  PROC DrawPart12()
    MoveL Offs(pOrigin,220.25,208.79,0.00),v40,z0,tPen\WObj:=wPaper;
    MoveL Offs(pOrigin,220.46,209.85,0.00),v40,fine,tPen\WObj:=wPaper;
    MoveL Offs(pOrigin,220.46,209.85,6.00),v60,z5,tPen\WObj:=wPaper;
    MoveL Offs(pOrigin,220.04,211.98,6.00),vTravel,z5,tPen\WObj:=wPaper;
    MoveL Offs(pOrigin,220.04,211.98,0.00),v60,z0,tPen\WObj:=wPaper;
    MoveL Offs(pOrigin,218.55,213.11,0.00),v40,z0,tPen\WObj:=wPaper;
    MoveL Offs(pOrigin,217.27,213.53,0.00),v40,z0,tPen\WObj:=wPaper;
    MoveL Offs(pOrigin,216.64,214.74,0.00),v40,z0,tPen\WObj:=wPaper;
    MoveL Offs(pOrigin,212.39,219.62,0.00),v40,z0,tPen\WObj:=wPaper;
    MoveL Offs(pOrigin,210.40,223.02,0.00),v40,z0,tPen\WObj:=wPaper;
    MoveL Offs(pOrigin,208.35,227.70,0.00),v40,fine,tPen\WObj:=wPaper;
    MoveL Offs(pOrigin,208.35,227.70,6.00),v60,z5,tPen\WObj:=wPaper;
    MoveL Offs(pOrigin,209.84,224.09,6.00),vTravel,z5,tPen\WObj:=wPaper;
    MoveL Offs(pOrigin,209.84,224.09,0.00),v60,z0,tPen\WObj:=wPaper;
    MoveL Offs(pOrigin,209.62,224.51,0.00),v40,z0,tPen\WObj:=wPaper;
    MoveL Offs(pOrigin,209.84,224.09,0.00),v40,fine,tPen\WObj:=wPaper;
    MoveL Offs(pOrigin,209.84,224.09,6.00),v60,z5,tPen\WObj:=wPaper;
    MoveL Offs(pOrigin,211.32,221.11,6.00),vTravel,z5,tPen\WObj:=wPaper;
    MoveL Offs(pOrigin,211.32,221.11,0.00),v60,z0,tPen\WObj:=wPaper;
    MoveL Offs(pOrigin,211.11,221.54,0.00),v40,z0,tPen\WObj:=wPaper;
    MoveL Offs(pOrigin,211.32,221.11,0.00),v40,fine,tPen\WObj:=wPaper;
    MoveL Offs(pOrigin,211.32,221.11,6.00),v60,z5,tPen\WObj:=wPaper;
    MoveL Offs(pOrigin,217.06,213.46,6.00),vTravel,z5,tPen\WObj:=wPaper;
    MoveL Offs(pOrigin,217.06,213.46,0.00),v60,z0,tPen\WObj:=wPaper;
    MoveL Offs(pOrigin,216.43,212.82,0.00),v40,fine,tPen\WObj:=wPaper;
    MoveL Offs(pOrigin,216.43,212.82,6.00),v60,z5,tPen\WObj:=wPaper;
    MoveL Offs(pOrigin,220.04,211.98,6.00),vTravel,z5,tPen\WObj:=wPaper;
    MoveL Offs(pOrigin,220.04,211.98,0.00),v60,z0,tPen\WObj:=wPaper;
    MoveL Offs(pOrigin,221.74,211.62,0.00),v40,z0,tPen\WObj:=wPaper;
    MoveL Offs(pOrigin,226.62,209.21,0.00),v40,fine,tPen\WObj:=wPaper;
    MoveL Offs(pOrigin,226.62,209.21,6.00),v60,z5,tPen\WObj:=wPaper;
    MoveL Offs(pOrigin,223.44,207.51,6.00),vTravel,z5,tPen\WObj:=wPaper;
    MoveL Offs(pOrigin,223.44,207.51,0.00),v60,z0,tPen\WObj:=wPaper;
    MoveL Offs(pOrigin,221.95,209.00,0.00),v40,z0,tPen\WObj:=wPaper;
    MoveL Offs(pOrigin,223.44,207.51,0.00),v40,fine,tPen\WObj:=wPaper;
    MoveL Offs(pOrigin,223.44,207.51,6.00),v60,z5,tPen\WObj:=wPaper;
    MoveL Offs(pOrigin,225.35,205.60,6.00),vTravel,z5,tPen\WObj:=wPaper;
    MoveL Offs(pOrigin,225.35,205.60,0.00),v60,z0,tPen\WObj:=wPaper;
    MoveL Offs(pOrigin,223.65,207.30,0.00),v40,z0,tPen\WObj:=wPaper;
    MoveL Offs(pOrigin,225.35,205.60,0.00),v40,fine,tPen\WObj:=wPaper;
    MoveL Offs(pOrigin,225.35,205.60,6.00),v60,z5,tPen\WObj:=wPaper;
    MoveL Offs(pOrigin,227.05,203.69,6.00),vTravel,z5,tPen\WObj:=wPaper;
    MoveL Offs(pOrigin,227.05,203.69,0.00),v60,z0,tPen\WObj:=wPaper;
    MoveL Offs(pOrigin,221.67,209.57,0.00),v40,z0,tPen\WObj:=wPaper;
    MoveL Offs(pOrigin,220.53,210.06,0.00),v40,z0,tPen\WObj:=wPaper;
    MoveL Offs(pOrigin,220.04,210.91,0.00),v40,z0,tPen\WObj:=wPaper;
    MoveL Offs(pOrigin,220.04,211.98,0.00),v40,fine,tPen\WObj:=wPaper;
    MoveL Offs(pOrigin,220.04,211.98,6.00),v60,z5,tPen\WObj:=wPaper;
    MoveL Offs(pOrigin,213.52,208.93,6.00),vTravel,z5,tPen\WObj:=wPaper;
    MoveL Offs(pOrigin,213.52,208.93,0.00),v60,z0,tPen\WObj:=wPaper;
    MoveL Offs(pOrigin,215.57,210.91,0.00),v40,z0,tPen\WObj:=wPaper;
    MoveL Offs(pOrigin,213.52,208.93,0.00),v40,fine,tPen\WObj:=wPaper;
    MoveL Offs(pOrigin,213.52,208.93,6.00),v60,z5,tPen\WObj:=wPaper;
    MoveL Offs(pOrigin,210.69,206.88,6.00),vTravel,z5,tPen\WObj:=wPaper;
    MoveL Offs(pOrigin,210.69,206.88,0.00),v60,z0,tPen\WObj:=wPaper;
    MoveL Offs(pOrigin,210.26,205.18,0.00),v40,z0,tPen\WObj:=wPaper;
    MoveL Offs(pOrigin,197.94,190.73,0.00),v40,z0,tPen\WObj:=wPaper;
    MoveL Offs(pOrigin,197.51,189.88,0.00),v40,z0,tPen\WObj:=wPaper;
    MoveL Offs(pOrigin,197.73,189.24,0.00),v40,z0,tPen\WObj:=wPaper;
    MoveL Offs(pOrigin,207.93,185.41,0.00),v40,z0,tPen\WObj:=wPaper;
    MoveL Offs(pOrigin,208.77,185.41,0.00),v40,z0,tPen\WObj:=wPaper;
    MoveL Offs(pOrigin,213.24,188.18,0.00),v40,z0,tPen\WObj:=wPaper;
    MoveL Offs(pOrigin,220.68,194.98,0.00),v40,z0,tPen\WObj:=wPaper;
    MoveL Offs(pOrigin,222.38,195.82,0.00),v40,fine,tPen\WObj:=wPaper;
    MoveL Offs(pOrigin,222.38,195.82,6.00),v60,z5,tPen\WObj:=wPaper;
    MoveL Offs(pOrigin,217.13,191.50,6.00),vTravel,z5,tPen\WObj:=wPaper;
    MoveL Offs(pOrigin,217.13,191.50,0.00),v60,z0,tPen\WObj:=wPaper;
    MoveL Offs(pOrigin,218.98,193.27,0.00),v40,z0,tPen\WObj:=wPaper;
    MoveL Offs(pOrigin,217.13,191.50,0.00),v40,fine,tPen\WObj:=wPaper;
    MoveL Offs(pOrigin,217.13,191.50,6.00),v60,z5,tPen\WObj:=wPaper;
    MoveL Offs(pOrigin,215.36,189.88,6.00),vTravel,z5,tPen\WObj:=wPaper;
    MoveL Offs(pOrigin,215.36,189.88,0.00),v60,z0,tPen\WObj:=wPaper;
    MoveL Offs(pOrigin,216.21,190.73,0.00),v40,z0,tPen\WObj:=wPaper;
    MoveL Offs(pOrigin,215.36,189.88,0.00),v40,fine,tPen\WObj:=wPaper;
    MoveL Offs(pOrigin,215.36,189.88,6.00),v60,z5,tPen\WObj:=wPaper;
    MoveL Offs(pOrigin,207.93,185.20,6.00),vTravel,z5,tPen\WObj:=wPaper;
    MoveL Offs(pOrigin,207.93,185.20,0.00),v60,z0,tPen\WObj:=wPaper;
    MoveL Offs(pOrigin,207.50,184.56,0.00),v40,z0,tPen\WObj:=wPaper;
    MoveL Offs(pOrigin,195.60,178.26,0.00),v40,z0,tPen\WObj:=wPaper;
    MoveL Offs(pOrigin,194.68,177.55,0.00),v40,z0,tPen\WObj:=wPaper;
    MoveL Offs(pOrigin,194.54,176.49,0.00),v40,z0,tPen\WObj:=wPaper;
    MoveL Offs(pOrigin,201.76,148.65,0.00),v40,z0,tPen\WObj:=wPaper;
    MoveL Offs(pOrigin,207.07,129.74,0.00),v40,z0,tPen\WObj:=wPaper;
    MoveL Offs(pOrigin,208.14,124.85,0.00),v40,z0,tPen\WObj:=wPaper;
    MoveL Offs(pOrigin,207.71,123.36,0.00),v40,z0,tPen\WObj:=wPaper;
    MoveL Offs(pOrigin,207.71,121.66,0.00),v40,z0,tPen\WObj:=wPaper;
    MoveL Offs(pOrigin,208.77,114.01,0.00),v40,z0,tPen\WObj:=wPaper;
    MoveL Offs(pOrigin,210.48,95.53,0.00),v40,fine,tPen\WObj:=wPaper;
    MoveL Offs(pOrigin,210.48,95.53,6.00),v60,z5,tPen\WObj:=wPaper;
    MoveL Offs(pOrigin,230.02,83.20,6.00),vTravel,z5,tPen\WObj:=wPaper;
    MoveL Offs(pOrigin,230.02,83.20,0.00),v60,z0,tPen\WObj:=wPaper;
    MoveL Offs(pOrigin,230.95,82.56,0.00),v40,z0,tPen\WObj:=wPaper;
    MoveL Offs(pOrigin,233.57,77.46,0.00),v40,z0,tPen\WObj:=wPaper;
    MoveL Offs(pOrigin,236.82,73.00,0.00),v40,z0,tPen\WObj:=wPaper;
    MoveL Offs(pOrigin,236.40,73.43,0.00),v40,z0,tPen\WObj:=wPaper;
    MoveL Offs(pOrigin,236.19,73.85,0.00),v40,z0,tPen\WObj:=wPaper;
    MoveL Offs(pOrigin,236.40,73.43,0.00),v40,fine,tPen\WObj:=wPaper;
    MoveL Offs(pOrigin,236.40,73.43,6.00),v60,z5,tPen\WObj:=wPaper;
    MoveL Offs(pOrigin,235.34,63.22,6.00),vTravel,z5,tPen\WObj:=wPaper;
    MoveL Offs(pOrigin,235.34,63.22,0.00),v60,z0,tPen\WObj:=wPaper;
    MoveL Offs(pOrigin,230.88,66.06,0.00),v40,z0,tPen\WObj:=wPaper;
    MoveL Offs(pOrigin,227.69,67.26,0.00),v40,z0,tPen\WObj:=wPaper;
    MoveL Offs(pOrigin,226.84,67.26,0.00),v40,fine,tPen\WObj:=wPaper;
    MoveL Offs(pOrigin,226.84,67.26,6.00),v60,z5,tPen\WObj:=wPaper;
    MoveL Offs(pOrigin,226.62,65.99,6.00),vTravel,z5,tPen\WObj:=wPaper;
    MoveL Offs(pOrigin,226.62,65.99,0.00),v60,z0,tPen\WObj:=wPaper;
    MoveL Offs(pOrigin,228.04,64.71,0.00),v40,z0,tPen\WObj:=wPaper;
    MoveL Offs(pOrigin,235.12,54.09,0.00),v40,z0,tPen\WObj:=wPaper;
    MoveL Offs(pOrigin,234.70,54.51,0.00),v40,z0,tPen\WObj:=wPaper;
    MoveL Offs(pOrigin,234.49,54.94,0.00),v40,z0,tPen\WObj:=wPaper;
    MoveL Offs(pOrigin,234.70,54.51,0.00),v40,fine,tPen\WObj:=wPaper;
    MoveL Offs(pOrigin,234.70,54.51,6.00),v60,z5,tPen\WObj:=wPaper;
    MoveL Offs(pOrigin,238.74,39.85,6.00),vTravel,z5,tPen\WObj:=wPaper;
    MoveL Offs(pOrigin,238.74,39.85,0.00),v60,z0,tPen\WObj:=wPaper;
    MoveL Offs(pOrigin,242.14,39.64,0.00),v40,z0,tPen\WObj:=wPaper;
    MoveL Offs(pOrigin,242.14,39.64,0.00),v40,z0,tPen\WObj:=wPaper;
    MoveL Offs(pOrigin,241.93,37.30,0.00),v40,z0,tPen\WObj:=wPaper;
    MoveL Offs(pOrigin,242.70,35.60,0.00),v40,z0,tPen\WObj:=wPaper;
    MoveL Offs(pOrigin,243.62,34.82,0.00),v40,z0,tPen\WObj:=wPaper;
    MoveL Offs(pOrigin,244.69,34.75,0.00),v40,z0,tPen\WObj:=wPaper;
  ENDPROC

  PROC DrawPart13()
    MoveL Offs(pOrigin,244.69,34.75,0.00),v40,z0,tPen\WObj:=wPaper;
    MoveL Offs(pOrigin,245.25,36.24,0.00),v40,z0,tPen\WObj:=wPaper;
    MoveL Offs(pOrigin,246.81,38.15,0.00),v40,z0,tPen\WObj:=wPaper;
    MoveL Offs(pOrigin,254.25,44.10,0.00),v40,z0,tPen\WObj:=wPaper;
    MoveL Offs(pOrigin,264.45,51.18,0.00),v40,z0,tPen\WObj:=wPaper;
    MoveL Offs(pOrigin,270.19,53.80,0.00),v40,z0,tPen\WObj:=wPaper;
    MoveL Offs(pOrigin,270.61,54.30,0.00),v40,z0,tPen\WObj:=wPaper;
    MoveL Offs(pOrigin,270.61,54.30,0.00),v40,z0,tPen\WObj:=wPaper;
    MoveL Offs(pOrigin,269.62,57.28,0.00),v40,z0,tPen\WObj:=wPaper;
    MoveL Offs(pOrigin,268.20,59.40,0.00),v40,z0,tPen\WObj:=wPaper;
    MoveL Offs(pOrigin,266.36,61.10,0.00),v40,fine,tPen\WObj:=wPaper;
    MoveL Offs(pOrigin,266.36,61.10,6.00),v60,z5,tPen\WObj:=wPaper;
    MoveL Offs(pOrigin,267.42,61.74,6.00),vTravel,z5,tPen\WObj:=wPaper;
    MoveL Offs(pOrigin,267.42,61.74,0.00),v60,z0,tPen\WObj:=wPaper;
    MoveL Offs(pOrigin,269.12,59.83,0.00),v40,z0,tPen\WObj:=wPaper;
    MoveL Offs(pOrigin,270.68,57.28,0.00),v40,z0,tPen\WObj:=wPaper;
    MoveL Offs(pOrigin,271.25,54.94,0.00),v40,z0,tPen\WObj:=wPaper;
    MoveL Offs(pOrigin,270.61,54.30,0.00),v40,z0,tPen\WObj:=wPaper;
    MoveL Offs(pOrigin,271.25,54.51,0.00),v40,z0,tPen\WObj:=wPaper;
    MoveL Offs(pOrigin,272.10,54.51,0.00),v40,z0,tPen\WObj:=wPaper;
    MoveL Offs(pOrigin,273.16,55.15,0.00),v40,z0,tPen\WObj:=wPaper;
    MoveL Offs(pOrigin,273.16,55.15,0.00),v40,z0,tPen\WObj:=wPaper;
    MoveL Offs(pOrigin,271.11,59.83,0.00),v40,z0,tPen\WObj:=wPaper;
    MoveL Offs(pOrigin,269.55,61.31,0.00),v40,fine,tPen\WObj:=wPaper;
    MoveL Offs(pOrigin,269.55,61.31,6.00),v60,z5,tPen\WObj:=wPaper;
    MoveL Offs(pOrigin,271.04,61.31,6.00),vTravel,z5,tPen\WObj:=wPaper;
    MoveL Offs(pOrigin,271.04,61.31,0.00),v60,z0,tPen\WObj:=wPaper;
    MoveL Offs(pOrigin,270.83,61.74,0.00),v40,z0,tPen\WObj:=wPaper;
    MoveL Offs(pOrigin,271.04,61.31,0.00),v40,z0,tPen\WObj:=wPaper;
    MoveL Offs(pOrigin,271.67,60.67,0.00),v40,z0,tPen\WObj:=wPaper;
    MoveL Offs(pOrigin,271.46,61.10,0.00),v40,z0,tPen\WObj:=wPaper;
    MoveL Offs(pOrigin,271.67,60.67,0.00),v40,fine,tPen\WObj:=wPaper;
    MoveL Offs(pOrigin,271.67,60.67,6.00),v60,z5,tPen\WObj:=wPaper;
    MoveL Offs(pOrigin,272.31,59.61,6.00),vTravel,z5,tPen\WObj:=wPaper;
    MoveL Offs(pOrigin,272.31,59.61,0.00),v60,z0,tPen\WObj:=wPaper;
    MoveL Offs(pOrigin,272.10,60.04,0.00),v40,z0,tPen\WObj:=wPaper;
    MoveL Offs(pOrigin,272.31,59.61,0.00),v40,fine,tPen\WObj:=wPaper;
    MoveL Offs(pOrigin,272.31,59.61,6.00),v60,z5,tPen\WObj:=wPaper;
    MoveL Offs(pOrigin,270.61,57.06,6.00),vTravel,z5,tPen\WObj:=wPaper;
    MoveL Offs(pOrigin,270.61,57.06,0.00),v60,z0,tPen\WObj:=wPaper;
    MoveL Offs(pOrigin,270.40,57.49,0.00),v40,z0,tPen\WObj:=wPaper;
    MoveL Offs(pOrigin,270.61,57.06,0.00),v40,z0,tPen\WObj:=wPaper;
    MoveL Offs(pOrigin,269.55,57.06,0.00),v40,z0,tPen\WObj:=wPaper;
    MoveL Offs(pOrigin,269.34,57.49,0.00),v40,z0,tPen\WObj:=wPaper;
    MoveL Offs(pOrigin,269.55,57.06,0.00),v40,fine,tPen\WObj:=wPaper;
    MoveL Offs(pOrigin,269.55,57.06,6.00),v60,z5,tPen\WObj:=wPaper;
    MoveL Offs(pOrigin,267.85,59.83,6.00),vTravel,z5,tPen\WObj:=wPaper;
    MoveL Offs(pOrigin,267.85,59.83,0.00),v60,z0,tPen\WObj:=wPaper;
    MoveL Offs(pOrigin,268.06,59.40,0.00),v40,z0,tPen\WObj:=wPaper;
    MoveL Offs(pOrigin,267.85,59.83,0.00),v40,fine,tPen\WObj:=wPaper;
    MoveL Offs(pOrigin,267.85,59.83,6.00),v60,z5,tPen\WObj:=wPaper;
    MoveL Offs(pOrigin,270.19,62.80,6.00),vTravel,z5,tPen\WObj:=wPaper;
    MoveL Offs(pOrigin,270.19,62.80,0.00),v60,z0,tPen\WObj:=wPaper;
    MoveL Offs(pOrigin,268.27,62.45,0.00),v40,z0,tPen\WObj:=wPaper;
    MoveL Offs(pOrigin,266.15,61.17,0.00),v40,z0,tPen\WObj:=wPaper;
    MoveL Offs(pOrigin,264.24,60.53,0.00),v40,z0,tPen\WObj:=wPaper;
    MoveL Offs(pOrigin,261.26,59.05,0.00),v40,z0,tPen\WObj:=wPaper;
    MoveL Offs(pOrigin,257.86,56.64,0.00),v40,z0,tPen\WObj:=wPaper;
    MoveL Offs(pOrigin,248.94,47.92,0.00),v40,z0,tPen\WObj:=wPaper;
    MoveL Offs(pOrigin,245.32,43.67,0.00),v40,z0,tPen\WObj:=wPaper;
    MoveL Offs(pOrigin,242.77,40.06,0.00),v40,z0,tPen\WObj:=wPaper;
    MoveL Offs(pOrigin,242.14,39.64,0.00),v40,fine,tPen\WObj:=wPaper;
    MoveL Offs(pOrigin,242.14,39.64,6.00),v60,z5,tPen\WObj:=wPaper;
    MoveL Offs(pOrigin,246.18,37.30,6.00),vTravel,z5,tPen\WObj:=wPaper;
    MoveL Offs(pOrigin,246.18,37.30,0.00),v60,z0,tPen\WObj:=wPaper;
    MoveL Offs(pOrigin,247.02,38.15,0.00),v40,z0,tPen\WObj:=wPaper;
    MoveL Offs(pOrigin,246.18,37.30,0.00),v40,fine,tPen\WObj:=wPaper;
    MoveL Offs(pOrigin,246.18,37.30,6.00),v60,z5,tPen\WObj:=wPaper;
    MoveL Offs(pOrigin,247.88,38.79,6.00),vTravel,z5,tPen\WObj:=wPaper;
    MoveL Offs(pOrigin,247.88,38.79,0.00),v60,z0,tPen\WObj:=wPaper;
    MoveL Offs(pOrigin,248.30,39.21,0.00),v40,z0,tPen\WObj:=wPaper;
    MoveL Offs(pOrigin,247.88,38.79,0.00),v40,fine,tPen\WObj:=wPaper;
    MoveL Offs(pOrigin,247.88,38.79,6.00),v60,z5,tPen\WObj:=wPaper;
    MoveL Offs(pOrigin,249.15,39.85,6.00),vTravel,z5,tPen\WObj:=wPaper;
    MoveL Offs(pOrigin,249.15,39.85,0.00),v60,z0,tPen\WObj:=wPaper;
    MoveL Offs(pOrigin,250.00,40.70,0.00),v40,z0,tPen\WObj:=wPaper;
    MoveL Offs(pOrigin,249.15,39.85,0.00),v40,fine,tPen\WObj:=wPaper;
    MoveL Offs(pOrigin,249.15,39.85,6.00),v60,z5,tPen\WObj:=wPaper;
    MoveL Offs(pOrigin,244.69,34.75,6.00),vTravel,z5,tPen\WObj:=wPaper;
    MoveL Offs(pOrigin,244.69,34.75,0.00),v60,z0,tPen\WObj:=wPaper;
    MoveL Offs(pOrigin,244.69,33.47,0.00),v40,z0,tPen\WObj:=wPaper;
    MoveL Offs(pOrigin,245.75,31.42,0.00),v40,z0,tPen\WObj:=wPaper;
    MoveL Offs(pOrigin,247.45,30.50,0.00),v40,z0,tPen\WObj:=wPaper;
    MoveL Offs(pOrigin,249.79,30.50,0.00),v40,z0,tPen\WObj:=wPaper;
    MoveL Offs(pOrigin,250.43,30.08,0.00),v40,z0,tPen\WObj:=wPaper;
    MoveL Offs(pOrigin,250.43,30.08,0.00),v40,z0,tPen\WObj:=wPaper;
    MoveL Offs(pOrigin,249.57,29.15,0.00),v40,z0,tPen\WObj:=wPaper;
    MoveL Offs(pOrigin,215.15,21.79,0.00),v40,z0,tPen\WObj:=wPaper;
    MoveL Offs(pOrigin,211.54,20.51,0.00),v40,z0,tPen\WObj:=wPaper;
    MoveL Offs(pOrigin,210.05,20.73,0.00),v40,z0,tPen\WObj:=wPaper;
    MoveL Offs(pOrigin,210.05,20.73,0.00),v40,z0,tPen\WObj:=wPaper;
    MoveL Offs(pOrigin,210.05,21.15,0.00),v40,z0,tPen\WObj:=wPaper;
    MoveL Offs(pOrigin,209.41,21.36,0.00),v40,z0,tPen\WObj:=wPaper;
    MoveL Offs(pOrigin,208.56,20.94,0.00),v40,fine,tPen\WObj:=wPaper;
    MoveL Offs(pOrigin,208.56,20.94,6.00),v60,z5,tPen\WObj:=wPaper;
    MoveL Offs(pOrigin,210.05,20.73,6.00),vTravel,z5,tPen\WObj:=wPaper;
    MoveL Offs(pOrigin,210.05,20.73,0.00),v60,z0,tPen\WObj:=wPaper;
    MoveL Offs(pOrigin,208.99,18.39,0.00),v40,z0,tPen\WObj:=wPaper;
    MoveL Offs(pOrigin,209.06,17.33,0.00),v40,z0,tPen\WObj:=wPaper;
    MoveL Offs(pOrigin,209.41,17.11,0.00),v40,z0,tPen\WObj:=wPaper;
    MoveL Offs(pOrigin,233.43,14.99,0.00),v40,z0,tPen\WObj:=wPaper;
    MoveL Offs(pOrigin,274.86,25.83,0.00),v40,fine,tPen\WObj:=wPaper;
    MoveL Offs(pOrigin,274.86,25.83,6.00),v60,z5,tPen\WObj:=wPaper;
    MoveL Offs(pOrigin,273.80,27.74,6.00),vTravel,z5,tPen\WObj:=wPaper;
    MoveL Offs(pOrigin,273.80,27.74,0.00),v60,z0,tPen\WObj:=wPaper;
    MoveL Offs(pOrigin,234.27,17.96,0.00),v40,z0,tPen\WObj:=wPaper;
    MoveL Offs(pOrigin,231.30,17.96,0.00),v40,z0,tPen\WObj:=wPaper;
    MoveL Offs(pOrigin,212.60,19.88,0.00),v40,z0,tPen\WObj:=wPaper;
    MoveL Offs(pOrigin,211.96,20.51,0.00),v40,fine,tPen\WObj:=wPaper;
    MoveL Offs(pOrigin,211.96,20.51,6.00),v60,z5,tPen\WObj:=wPaper;
    MoveL Offs(pOrigin,208.99,17.11,6.00),vTravel,z5,tPen\WObj:=wPaper;
    MoveL Offs(pOrigin,208.99,17.11,0.00),v60,z0,tPen\WObj:=wPaper;
    MoveL Offs(pOrigin,208.77,16.26,0.00),v40,z0,tPen\WObj:=wPaper;
    MoveL Offs(pOrigin,209.41,14.35,0.00),v40,fine,tPen\WObj:=wPaper;
    MoveL Offs(pOrigin,209.41,14.35,6.00),v60,z5,tPen\WObj:=wPaper;
    MoveL Offs(pOrigin,207.07,13.93,6.00),vTravel,z5,tPen\WObj:=wPaper;
    MoveL Offs(pOrigin,207.07,13.93,0.00),v60,z0,tPen\WObj:=wPaper;
    MoveL Offs(pOrigin,208.99,13.78,0.00),v40,z0,tPen\WObj:=wPaper;
    MoveL Offs(pOrigin,209.84,14.35,0.00),v40,z0,tPen\WObj:=wPaper;
    MoveL Offs(pOrigin,212.81,14.35,0.00),v40,z0,tPen\WObj:=wPaper;
  ENDPROC

  PROC DrawPart14()
    MoveL Offs(pOrigin,232.15,12.23,0.00),v40,z0,tPen\WObj:=wPaper;
    MoveL Offs(pOrigin,235.12,12.44,0.00),v40,z0,tPen\WObj:=wPaper;
    MoveL Offs(pOrigin,276.35,23.27,0.00),v40,z0,tPen\WObj:=wPaper;
    MoveL Offs(pOrigin,276.56,23.70,0.00),v40,fine,tPen\WObj:=wPaper;
    MoveL Offs(pOrigin,276.56,23.70,6.00),v60,z5,tPen\WObj:=wPaper;
    MoveL Offs(pOrigin,273.59,29.01,6.00),vTravel,z5,tPen\WObj:=wPaper;
    MoveL Offs(pOrigin,273.59,29.01,0.00),v60,z0,tPen\WObj:=wPaper;
    MoveL Offs(pOrigin,272.31,29.01,0.00),v40,z0,tPen\WObj:=wPaper;
    MoveL Offs(pOrigin,271.89,29.44,0.00),v40,z0,tPen\WObj:=wPaper;
    MoveL Offs(pOrigin,271.89,29.44,0.00),v40,z0,tPen\WObj:=wPaper;
    MoveL Offs(pOrigin,272.31,30.08,0.00),v40,z0,tPen\WObj:=wPaper;
    MoveL Offs(pOrigin,273.59,30.08,0.00),v40,z0,tPen\WObj:=wPaper;
    MoveL Offs(pOrigin,273.59,30.08,0.00),v40,z0,tPen\WObj:=wPaper;
    MoveL Offs(pOrigin,274.01,30.50,0.00),v40,z0,tPen\WObj:=wPaper;
    MoveL Offs(pOrigin,282.94,33.62,0.00),v40,z0,tPen\WObj:=wPaper;
    MoveL Offs(pOrigin,285.91,35.39,0.00),v40,z0,tPen\WObj:=wPaper;
    MoveL Offs(pOrigin,285.91,35.39,0.00),v40,z0,tPen\WObj:=wPaper;
    MoveL Offs(pOrigin,287.83,35.74,0.00),v40,z0,tPen\WObj:=wPaper;
    MoveL Offs(pOrigin,288.25,36.45,0.00),v40,z0,tPen\WObj:=wPaper;
    MoveL Offs(pOrigin,288.46,36.45,0.00),v40,z0,tPen\WObj:=wPaper;
    MoveL Offs(pOrigin,290.80,37.37,0.00),v40,z0,tPen\WObj:=wPaper;
    MoveL Offs(pOrigin,291.51,38.36,0.00),v40,z0,tPen\WObj:=wPaper;
    MoveL Offs(pOrigin,291.65,39.42,0.00),v40,z0,tPen\WObj:=wPaper;
    MoveL Offs(pOrigin,289.60,45.59,0.00),v40,z0,tPen\WObj:=wPaper;
    MoveL Offs(pOrigin,288.67,46.22,0.00),v40,z0,tPen\WObj:=wPaper;
    MoveL Offs(pOrigin,287.61,46.22,0.00),v40,z0,tPen\WObj:=wPaper;
    MoveL Offs(pOrigin,284.42,45.02,0.00),v40,z0,tPen\WObj:=wPaper;
    MoveL Offs(pOrigin,283.79,44.10,0.00),v40,z0,tPen\WObj:=wPaper;
    MoveL Offs(pOrigin,285.70,39.21,0.00),v40,z0,tPen\WObj:=wPaper;
    MoveL Offs(pOrigin,285.98,36.88,0.00),v40,z0,tPen\WObj:=wPaper;
    MoveL Offs(pOrigin,288.46,36.45,0.00),v40,fine,tPen\WObj:=wPaper;
    MoveL Offs(pOrigin,288.46,36.45,6.00),v60,z5,tPen\WObj:=wPaper;
    MoveL Offs(pOrigin,287.40,38.58,6.00),vTravel,z5,tPen\WObj:=wPaper;
    MoveL Offs(pOrigin,287.40,38.58,0.00),v60,z0,tPen\WObj:=wPaper;
    MoveL Offs(pOrigin,285.49,43.25,0.00),v40,z0,tPen\WObj:=wPaper;
    MoveL Offs(pOrigin,286.12,43.96,0.00),v40,z0,tPen\WObj:=wPaper;
    MoveL Offs(pOrigin,288.46,44.74,0.00),v40,fine,tPen\WObj:=wPaper;
    MoveL Offs(pOrigin,288.46,44.74,6.00),v60,z5,tPen\WObj:=wPaper;
    MoveL Offs(pOrigin,287.19,46.22,6.00),vTravel,z5,tPen\WObj:=wPaper;
    MoveL Offs(pOrigin,287.19,46.22,0.00),v60,z0,tPen\WObj:=wPaper;
    MoveL Offs(pOrigin,285.91,47.29,0.00),v40,fine,tPen\WObj:=wPaper;
    MoveL Offs(pOrigin,285.91,47.29,6.00),v60,z5,tPen\WObj:=wPaper;
    MoveL Offs(pOrigin,288.67,48.56,6.00),vTravel,z5,tPen\WObj:=wPaper;
    MoveL Offs(pOrigin,288.67,48.56,0.00),v60,z0,tPen\WObj:=wPaper;
    MoveL Offs(pOrigin,287.61,48.42,0.00),v40,z0,tPen\WObj:=wPaper;
    MoveL Offs(pOrigin,285.06,47.08,0.00),v40,z0,tPen\WObj:=wPaper;
    MoveL Offs(pOrigin,283.36,46.79,0.00),v40,z0,tPen\WObj:=wPaper;
    MoveL Offs(pOrigin,282.09,45.80,0.00),v40,z0,tPen\WObj:=wPaper;
    MoveL Offs(pOrigin,282.09,45.80,0.00),v40,z0,tPen\WObj:=wPaper;
    MoveL Offs(pOrigin,283.36,44.74,0.00),v40,z0,tPen\WObj:=wPaper;
    MoveL Offs(pOrigin,283.79,44.74,0.00),v40,fine,tPen\WObj:=wPaper;
    MoveL Offs(pOrigin,283.79,44.74,6.00),v60,z5,tPen\WObj:=wPaper;
    MoveL Offs(pOrigin,284.21,42.83,6.00),vTravel,z5,tPen\WObj:=wPaper;
    MoveL Offs(pOrigin,284.21,42.83,0.00),v60,z0,tPen\WObj:=wPaper;
    MoveL Offs(pOrigin,284.00,43.25,0.00),v40,z0,tPen\WObj:=wPaper;
    MoveL Offs(pOrigin,284.21,42.83,0.00),v40,fine,tPen\WObj:=wPaper;
    MoveL Offs(pOrigin,284.21,42.83,6.00),v60,z5,tPen\WObj:=wPaper;
    MoveL Offs(pOrigin,286.98,42.40,6.00),vTravel,z5,tPen\WObj:=wPaper;
    MoveL Offs(pOrigin,286.98,42.40,0.00),v60,z0,tPen\WObj:=wPaper;
    MoveL Offs(pOrigin,287.40,41.55,0.00),v40,fine,tPen\WObj:=wPaper;
    MoveL Offs(pOrigin,287.40,41.55,6.00),v60,z5,tPen\WObj:=wPaper;
    MoveL Offs(pOrigin,289.95,41.76,6.00),vTravel,z5,tPen\WObj:=wPaper;
    MoveL Offs(pOrigin,289.95,41.76,0.00),v60,z0,tPen\WObj:=wPaper;
    MoveL Offs(pOrigin,290.09,39.42,0.00),v40,z0,tPen\WObj:=wPaper;
    MoveL Offs(pOrigin,288.46,39.00,0.00),v40,fine,tPen\WObj:=wPaper;
    MoveL Offs(pOrigin,288.46,39.00,6.00),v60,z5,tPen\WObj:=wPaper;
    MoveL Offs(pOrigin,291.01,37.30,6.00),vTravel,z5,tPen\WObj:=wPaper;
    MoveL Offs(pOrigin,291.01,37.30,0.00),v60,z0,tPen\WObj:=wPaper;
    MoveL Offs(pOrigin,292.50,37.51,0.00),v40,z0,tPen\WObj:=wPaper;
    MoveL Offs(pOrigin,294.41,38.36,0.00),v40,fine,tPen\WObj:=wPaper;
    MoveL Offs(pOrigin,294.41,38.36,6.00),v60,z5,tPen\WObj:=wPaper;
    MoveL Offs(pOrigin,285.91,36.66,6.00),vTravel,z5,tPen\WObj:=wPaper;
    MoveL Offs(pOrigin,285.91,36.66,0.00),v60,z0,tPen\WObj:=wPaper;
    MoveL Offs(pOrigin,285.91,35.39,0.00),v40,fine,tPen\WObj:=wPaper;
    MoveL Offs(pOrigin,285.91,35.39,6.00),v60,z5,tPen\WObj:=wPaper;
    MoveL Offs(pOrigin,282.09,45.80,6.00),vTravel,z5,tPen\WObj:=wPaper;
    MoveL Offs(pOrigin,282.09,45.80,0.00),v60,z0,tPen\WObj:=wPaper;
    MoveL Offs(pOrigin,279.54,45.38,0.00),v40,z0,tPen\WObj:=wPaper;
    MoveL Offs(pOrigin,276.77,44.38,0.00),v40,z0,tPen\WObj:=wPaper;
    MoveL Offs(pOrigin,260.62,36.52,0.00),v40,z0,tPen\WObj:=wPaper;
    MoveL Offs(pOrigin,255.10,32.84,0.00),v40,z0,tPen\WObj:=wPaper;
    MoveL Offs(pOrigin,254.68,31.77,0.00),v40,z0,tPen\WObj:=wPaper;
    MoveL Offs(pOrigin,254.68,31.77,0.00),v40,z0,tPen\WObj:=wPaper;
    MoveL Offs(pOrigin,254.89,30.29,0.00),v40,z0,tPen\WObj:=wPaper;
    MoveL Offs(pOrigin,255.95,29.23,0.00),v40,z0,tPen\WObj:=wPaper;
    MoveL Offs(pOrigin,257.44,28.59,0.00),v40,z0,tPen\WObj:=wPaper;
    MoveL Offs(pOrigin,264.24,28.38,0.00),v40,z0,tPen\WObj:=wPaper;
    MoveL Offs(pOrigin,269.98,29.44,0.00),v40,z0,tPen\WObj:=wPaper;
    MoveL Offs(pOrigin,271.89,29.44,0.00),v40,fine,tPen\WObj:=wPaper;
    MoveL Offs(pOrigin,271.89,29.44,6.00),v60,z5,tPen\WObj:=wPaper;
    MoveL Offs(pOrigin,273.59,30.08,6.00),vTravel,z5,tPen\WObj:=wPaper;
    MoveL Offs(pOrigin,273.59,30.08,0.00),v60,z0,tPen\WObj:=wPaper;
    MoveL Offs(pOrigin,273.80,28.16,0.00),v40,z0,tPen\WObj:=wPaper;
    MoveL Offs(pOrigin,274.86,26.04,0.00),v40,z0,tPen\WObj:=wPaper;
    MoveL Offs(pOrigin,276.77,23.77,0.00),v40,z0,tPen\WObj:=wPaper;
    MoveL Offs(pOrigin,278.05,23.49,0.00),v40,z0,tPen\WObj:=wPaper;
    MoveL Offs(pOrigin,284.85,23.70,0.00),v40,z0,tPen\WObj:=wPaper;
    MoveL Offs(pOrigin,293.99,25.83,0.00),v40,z0,tPen\WObj:=wPaper;
    MoveL Offs(pOrigin,295.05,27.03,0.00),v40,z0,tPen\WObj:=wPaper;
    MoveL Offs(pOrigin,298.02,28.59,0.00),v40,fine,tPen\WObj:=wPaper;
    MoveL Offs(pOrigin,298.02,28.59,6.00),v60,z5,tPen\WObj:=wPaper;
    MoveL Offs(pOrigin,294.41,25.83,6.00),vTravel,z5,tPen\WObj:=wPaper;
    MoveL Offs(pOrigin,294.41,25.83,0.00),v60,z0,tPen\WObj:=wPaper;
    MoveL Offs(pOrigin,297.17,25.19,0.00),v40,z0,tPen\WObj:=wPaper;
    MoveL Offs(pOrigin,302.91,25.19,0.00),v40,z0,tPen\WObj:=wPaper;
    MoveL Offs(pOrigin,306.74,25.83,0.00),v40,z0,tPen\WObj:=wPaper;
    MoveL Offs(pOrigin,311.84,27.52,0.00),v40,z0,tPen\WObj:=wPaper;
    MoveL Offs(pOrigin,313.96,27.81,0.00),v40,z0,tPen\WObj:=wPaper;
    MoveL Offs(pOrigin,314.46,28.80,0.00),v40,z0,tPen\WObj:=wPaper;
    MoveL Offs(pOrigin,315.45,29.51,0.00),v40,z0,tPen\WObj:=wPaper;
    MoveL Offs(pOrigin,321.97,32.20,0.00),v40,z0,tPen\WObj:=wPaper;
    MoveL Offs(pOrigin,323.52,36.24,0.00),v40,z0,tPen\WObj:=wPaper;
    MoveL Offs(pOrigin,324.16,40.28,0.00),v40,z0,tPen\WObj:=wPaper;
    MoveL Offs(pOrigin,324.16,42.61,0.00),v40,z0,tPen\WObj:=wPaper;
    MoveL Offs(pOrigin,322.89,50.26,0.00),v40,z0,tPen\WObj:=wPaper;
    MoveL Offs(pOrigin,320.98,54.51,0.00),v40,z0,tPen\WObj:=wPaper;
    MoveL Offs(pOrigin,320.98,54.51,0.00),v40,z0,tPen\WObj:=wPaper;
    MoveL Offs(pOrigin,320.90,55.58,0.00),v40,z0,tPen\WObj:=wPaper;
    MoveL Offs(pOrigin,318.64,58.97,0.00),v40,z0,tPen\WObj:=wPaper;
    MoveL Offs(pOrigin,316.94,60.53,0.00),v40,z0,tPen\WObj:=wPaper;
  ENDPROC

  PROC DrawPart15()
    MoveL Offs(pOrigin,314.60,61.38,0.00),v40,z0,tPen\WObj:=wPaper;
    MoveL Offs(pOrigin,313.96,62.30,0.00),v40,z0,tPen\WObj:=wPaper;
    MoveL Offs(pOrigin,311.41,62.80,0.00),v40,z0,tPen\WObj:=wPaper;
    MoveL Offs(pOrigin,310.14,63.44,0.00),v40,z0,tPen\WObj:=wPaper;
    MoveL Offs(pOrigin,306.52,63.44,0.00),v40,z0,tPen\WObj:=wPaper;
    MoveL Offs(pOrigin,302.49,62.30,0.00),v40,z0,tPen\WObj:=wPaper;
    MoveL Offs(pOrigin,301.85,61.31,0.00),v40,z0,tPen\WObj:=wPaper;
    MoveL Offs(pOrigin,301.85,61.31,0.00),v40,z0,tPen\WObj:=wPaper;
    MoveL Offs(pOrigin,302.49,60.67,0.00),v40,z0,tPen\WObj:=wPaper;
    MoveL Offs(pOrigin,305.67,60.32,0.00),v40,z0,tPen\WObj:=wPaper;
    MoveL Offs(pOrigin,310.56,61.10,0.00),v40,z0,tPen\WObj:=wPaper;
    MoveL Offs(pOrigin,310.56,61.10,0.00),v40,z0,tPen\WObj:=wPaper;
    MoveL Offs(pOrigin,313.75,60.89,0.00),v40,z0,tPen\WObj:=wPaper;
    MoveL Offs(pOrigin,313.75,60.89,0.00),v40,z0,tPen\WObj:=wPaper;
    MoveL Offs(pOrigin,314.17,60.04,0.00),v40,z0,tPen\WObj:=wPaper;
    MoveL Offs(pOrigin,316.30,58.76,0.00),v40,z0,tPen\WObj:=wPaper;
    MoveL Offs(pOrigin,318.64,56.42,0.00),v40,z0,tPen\WObj:=wPaper;
    MoveL Offs(pOrigin,320.34,54.30,0.00),v40,fine,tPen\WObj:=wPaper;
    MoveL Offs(pOrigin,320.34,54.30,6.00),v60,z5,tPen\WObj:=wPaper;
    MoveL Offs(pOrigin,319.27,53.45,6.00),vTravel,z5,tPen\WObj:=wPaper;
    MoveL Offs(pOrigin,319.27,53.45,0.00),v60,z0,tPen\WObj:=wPaper;
    MoveL Offs(pOrigin,319.06,53.88,0.00),v40,z0,tPen\WObj:=wPaper;
    MoveL Offs(pOrigin,319.27,53.45,0.00),v40,fine,tPen\WObj:=wPaper;
    MoveL Offs(pOrigin,319.27,53.45,6.00),v60,z5,tPen\WObj:=wPaper;
    MoveL Offs(pOrigin,317.58,56.00,6.00),vTravel,z5,tPen\WObj:=wPaper;
    MoveL Offs(pOrigin,317.58,56.00,0.00),v60,z0,tPen\WObj:=wPaper;
    MoveL Offs(pOrigin,317.36,56.42,0.00),v40,z0,tPen\WObj:=wPaper;
    MoveL Offs(pOrigin,317.58,56.00,0.00),v40,z0,tPen\WObj:=wPaper;
    MoveL Offs(pOrigin,317.36,56.42,0.00),v40,z0,tPen\WObj:=wPaper;
    MoveL Offs(pOrigin,319.35,53.66,0.00),v40,z0,tPen\WObj:=wPaper;
    MoveL Offs(pOrigin,321.26,49.62,0.00),v40,z0,tPen\WObj:=wPaper;
    MoveL Offs(pOrigin,322.67,44.10,0.00),v40,z0,tPen\WObj:=wPaper;
    MoveL Offs(pOrigin,322.67,40.49,0.00),v40,fine,tPen\WObj:=wPaper;
    MoveL Offs(pOrigin,322.67,40.49,6.00),v60,z5,tPen\WObj:=wPaper;
    MoveL Offs(pOrigin,322.04,31.99,6.00),vTravel,z5,tPen\WObj:=wPaper;
    MoveL Offs(pOrigin,322.04,31.99,0.00),v60,z0,tPen\WObj:=wPaper;
    MoveL Offs(pOrigin,321.68,30.08,0.00),v40,z0,tPen\WObj:=wPaper;
    MoveL Offs(pOrigin,320.12,28.16,0.00),v40,z0,tPen\WObj:=wPaper;
    MoveL Offs(pOrigin,316.73,26.89,0.00),v40,z0,tPen\WObj:=wPaper;
    MoveL Offs(pOrigin,316.73,26.89,0.00),v40,z0,tPen\WObj:=wPaper;
    MoveL Offs(pOrigin,317.58,25.83,0.00),v40,z0,tPen\WObj:=wPaper;
    MoveL Offs(pOrigin,320.98,25.61,0.00),v40,z0,tPen\WObj:=wPaper;
    MoveL Offs(pOrigin,333.94,27.74,0.00),v40,z0,tPen\WObj:=wPaper;
    MoveL Offs(pOrigin,335.00,27.52,0.00),v40,z0,tPen\WObj:=wPaper;
    MoveL Offs(pOrigin,335.00,27.52,0.00),v40,z0,tPen\WObj:=wPaper;
    MoveL Offs(pOrigin,335.85,26.39,0.00),v40,z0,tPen\WObj:=wPaper;
    MoveL Offs(pOrigin,339.25,25.19,0.00),v40,z0,tPen\WObj:=wPaper;
    MoveL Offs(pOrigin,345.41,24.76,0.00),v40,z0,tPen\WObj:=wPaper;
    MoveL Offs(pOrigin,349.88,25.97,0.00),v40,z0,tPen\WObj:=wPaper;
    MoveL Offs(pOrigin,359.86,30.36,0.00),v40,z0,tPen\WObj:=wPaper;
    MoveL Offs(pOrigin,365.60,32.20,0.00),v40,z0,tPen\WObj:=wPaper;
    MoveL Offs(pOrigin,365.60,32.20,0.00),v40,z0,tPen\WObj:=wPaper;
    MoveL Offs(pOrigin,366.24,31.77,0.00),v40,z0,tPen\WObj:=wPaper;
    MoveL Offs(pOrigin,385.79,34.33,0.00),v40,z0,tPen\WObj:=wPaper;
    MoveL Offs(pOrigin,397.26,36.66,0.00),v40,z0,tPen\WObj:=wPaper;
    MoveL Offs(pOrigin,403.85,38.72,0.00),v40,z0,tPen\WObj:=wPaper;
    MoveL Offs(pOrigin,407.46,40.42,0.00),v40,z0,tPen\WObj:=wPaper;
    MoveL Offs(pOrigin,411.08,43.25,0.00),v40,z0,tPen\WObj:=wPaper;
    MoveL Offs(pOrigin,412.85,45.80,0.00),v40,z0,tPen\WObj:=wPaper;
    MoveL Offs(pOrigin,414.69,50.26,0.00),v40,z0,tPen\WObj:=wPaper;
    MoveL Offs(pOrigin,415.54,54.09,0.00),v40,z0,tPen\WObj:=wPaper;
    MoveL Offs(pOrigin,415.75,57.70,0.00),v40,z0,tPen\WObj:=wPaper;
    MoveL Offs(pOrigin,414.69,64.71,0.00),v40,z0,tPen\WObj:=wPaper;
    MoveL Offs(pOrigin,415.11,66.62,0.00),v40,z0,tPen\WObj:=wPaper;
    MoveL Offs(pOrigin,415.11,69.81,0.00),v40,z0,tPen\WObj:=wPaper;
    MoveL Offs(pOrigin,414.26,73.43,0.00),v40,z0,tPen\WObj:=wPaper;
    MoveL Offs(pOrigin,410.01,84.47,0.00),v40,z0,tPen\WObj:=wPaper;
    MoveL Offs(pOrigin,408.10,92.55,0.00),v40,z0,tPen\WObj:=wPaper;
    MoveL Offs(pOrigin,406.47,97.65,0.00),v40,z0,tPen\WObj:=wPaper;
    MoveL Offs(pOrigin,404.77,101.05,0.00),v40,z0,tPen\WObj:=wPaper;
    MoveL Offs(pOrigin,401.02,106.15,0.00),v40,z0,tPen\WObj:=wPaper;
    MoveL Offs(pOrigin,400.88,108.06,0.00),v40,z0,tPen\WObj:=wPaper;
    MoveL Offs(pOrigin,399.67,111.89,0.00),v40,z0,tPen\WObj:=wPaper;
    MoveL Offs(pOrigin,396.34,117.20,0.00),v40,z0,tPen\WObj:=wPaper;
    MoveL Offs(pOrigin,395.77,119.54,0.00),v40,z0,tPen\WObj:=wPaper;
    MoveL Offs(pOrigin,395.99,125.28,0.00),v40,z0,tPen\WObj:=wPaper;
    MoveL Offs(pOrigin,395.70,126.34,0.00),v40,z0,tPen\WObj:=wPaper;
    MoveL Offs(pOrigin,394.71,127.47,0.00),v40,z0,tPen\WObj:=wPaper;
    MoveL Offs(pOrigin,393.44,127.82,0.00),v40,z0,tPen\WObj:=wPaper;
    MoveL Offs(pOrigin,393.44,127.82,0.00),v40,z0,tPen\WObj:=wPaper;
    MoveL Offs(pOrigin,393.44,130.59,0.00),v40,z0,tPen\WObj:=wPaper;
    MoveL Offs(pOrigin,389.40,169.26,0.00),v40,z0,tPen\WObj:=wPaper;
    MoveL Offs(pOrigin,386.00,209.43,0.00),v40,z0,tPen\WObj:=wPaper;
    MoveL Offs(pOrigin,384.94,218.56,0.00),v40,z0,tPen\WObj:=wPaper;
    MoveL Offs(pOrigin,383.66,224.73,0.00),v40,z0,tPen\WObj:=wPaper;
    MoveL Offs(pOrigin,382.03,229.40,0.00),v40,z0,tPen\WObj:=wPaper;
    MoveL Offs(pOrigin,380.26,232.59,0.00),v40,z0,tPen\WObj:=wPaper;
    MoveL Offs(pOrigin,378.14,234.93,0.00),v40,z0,tPen\WObj:=wPaper;
    MoveL Offs(pOrigin,377.36,233.86,0.00),v40,z0,tPen\WObj:=wPaper;
    MoveL Offs(pOrigin,379.84,227.70,0.00),v40,z0,tPen\WObj:=wPaper;
    MoveL Offs(pOrigin,380.69,222.60,0.00),v40,z0,tPen\WObj:=wPaper;
    MoveL Offs(pOrigin,381.11,217.71,0.00),v40,z0,tPen\WObj:=wPaper;
    MoveL Offs(pOrigin,381.11,208.57,0.00),v40,z0,tPen\WObj:=wPaper;
    MoveL Offs(pOrigin,380.26,198.38,0.00),v40,z0,tPen\WObj:=wPaper;
    MoveL Offs(pOrigin,378.56,185.62,0.00),v40,z0,tPen\WObj:=wPaper;
    MoveL Offs(pOrigin,377.50,184.35,0.00),v40,z0,tPen\WObj:=wPaper;
    MoveL Offs(pOrigin,378.77,177.34,0.00),v40,z0,tPen\WObj:=wPaper;
    MoveL Offs(pOrigin,380.90,171.18,0.00),v40,z0,tPen\WObj:=wPaper;
    MoveL Offs(pOrigin,380.90,169.48,0.00),v40,z0,tPen\WObj:=wPaper;
    MoveL Offs(pOrigin,379.77,165.44,0.00),v40,z0,tPen\WObj:=wPaper;
    MoveL Offs(pOrigin,381.68,159.70,0.00),v40,z0,tPen\WObj:=wPaper;
    MoveL Offs(pOrigin,385.01,152.90,0.00),v40,z0,tPen\WObj:=wPaper;
    MoveL Offs(pOrigin,386.21,149.50,0.00),v40,z0,tPen\WObj:=wPaper;
    MoveL Offs(pOrigin,386.21,146.31,0.00),v40,z0,tPen\WObj:=wPaper;
    MoveL Offs(pOrigin,385.79,144.40,0.00),v40,z0,tPen\WObj:=wPaper;
    MoveL Offs(pOrigin,385.79,144.40,0.00),v40,z0,tPen\WObj:=wPaper;
    MoveL Offs(pOrigin,384.09,143.76,0.00),v40,z0,tPen\WObj:=wPaper;
    MoveL Offs(pOrigin,377.08,138.24,0.00),v40,z0,tPen\WObj:=wPaper;
    MoveL Offs(pOrigin,373.04,134.62,0.00),v40,fine,tPen\WObj:=wPaper;
    MoveL Offs(pOrigin,373.04,134.62,6.00),v60,z5,tPen\WObj:=wPaper;
    MoveL Offs(pOrigin,375.59,136.75,6.00),vTravel,z5,tPen\WObj:=wPaper;
    MoveL Offs(pOrigin,375.59,136.75,0.00),v60,z0,tPen\WObj:=wPaper;
    MoveL Offs(pOrigin,376.01,137.18,0.00),v40,z0,tPen\WObj:=wPaper;
    MoveL Offs(pOrigin,375.59,136.75,0.00),v40,fine,tPen\WObj:=wPaper;
    MoveL Offs(pOrigin,375.59,136.75,6.00),v60,z5,tPen\WObj:=wPaper;
    MoveL Offs(pOrigin,376.44,134.41,6.00),vTravel,z5,tPen\WObj:=wPaper;
    MoveL Offs(pOrigin,376.44,134.41,0.00),v60,z0,tPen\WObj:=wPaper;
    MoveL Offs(pOrigin,382.39,136.96,0.00),v40,z0,tPen\WObj:=wPaper;
    MoveL Offs(pOrigin,385.36,137.60,0.00),v40,z0,tPen\WObj:=wPaper;
    MoveL Offs(pOrigin,386.85,137.39,0.00),v40,fine,tPen\WObj:=wPaper;
  ENDPROC

  PROC DrawPart16()
    MoveL Offs(pOrigin,386.85,137.39,6.00),v60,z5,tPen\WObj:=wPaper;
    MoveL Offs(pOrigin,385.79,144.40,6.00),vTravel,z5,tPen\WObj:=wPaper;
    MoveL Offs(pOrigin,385.79,144.40,0.00),v60,z0,tPen\WObj:=wPaper;
    MoveL Offs(pOrigin,388.76,141.00,0.00),v40,z0,tPen\WObj:=wPaper;
    MoveL Offs(pOrigin,389.83,138.24,0.00),v40,z0,tPen\WObj:=wPaper;
    MoveL Offs(pOrigin,390.25,129.74,0.00),v40,z0,tPen\WObj:=wPaper;
    MoveL Offs(pOrigin,390.89,127.82,0.00),v40,fine,tPen\WObj:=wPaper;
    MoveL Offs(pOrigin,390.89,127.82,6.00),v60,z5,tPen\WObj:=wPaper;
    MoveL Offs(pOrigin,393.44,127.82,6.00),vTravel,z5,tPen\WObj:=wPaper;
    MoveL Offs(pOrigin,393.44,127.82,0.00),v60,z0,tPen\WObj:=wPaper;
    MoveL Offs(pOrigin,391.31,127.82,0.00),v40,z0,tPen\WObj:=wPaper;
    MoveL Offs(pOrigin,390.25,127.19,0.00),v40,z0,tPen\WObj:=wPaper;
    MoveL Offs(pOrigin,379.41,124.64,0.00),v40,fine,tPen\WObj:=wPaper;
    MoveL Offs(pOrigin,379.41,124.64,6.00),v60,z5,tPen\WObj:=wPaper;
    MoveL Offs(pOrigin,387.27,123.15,6.00),vTravel,z5,tPen\WObj:=wPaper;
    MoveL Offs(pOrigin,387.27,123.15,0.00),v60,z0,tPen\WObj:=wPaper;
    MoveL Offs(pOrigin,384.09,122.37,0.00),v40,z0,tPen\WObj:=wPaper;
    MoveL Offs(pOrigin,379.62,120.46,0.00),v40,z0,tPen\WObj:=wPaper;
    MoveL Offs(pOrigin,366.45,113.87,0.00),v40,z0,tPen\WObj:=wPaper;
    MoveL Offs(pOrigin,357.52,108.49,0.00),v40,z0,tPen\WObj:=wPaper;
    MoveL Offs(pOrigin,353.06,105.09,0.00),v40,z0,tPen\WObj:=wPaper;
    MoveL Offs(pOrigin,350.09,102.11,0.00),v40,z0,tPen\WObj:=wPaper;
    MoveL Offs(pOrigin,348.60,101.47,0.00),v40,z0,tPen\WObj:=wPaper;
    MoveL Offs(pOrigin,348.17,101.90,0.00),v40,z0,tPen\WObj:=wPaper;
    MoveL Offs(pOrigin,348.39,105.30,0.00),v40,z0,tPen\WObj:=wPaper;
    MoveL Offs(pOrigin,348.17,105.72,0.00),v40,z0,tPen\WObj:=wPaper;
    MoveL Offs(pOrigin,348.17,105.72,0.00),v40,z0,tPen\WObj:=wPaper;
    MoveL Offs(pOrigin,349.02,108.91,0.00),v40,z0,tPen\WObj:=wPaper;
    MoveL Offs(pOrigin,349.02,108.91,0.00),v40,z0,tPen\WObj:=wPaper;
    MoveL Offs(pOrigin,348.81,109.76,0.00),v40,z0,tPen\WObj:=wPaper;
    MoveL Offs(pOrigin,349.24,112.31,0.00),v40,z0,tPen\WObj:=wPaper;
    MoveL Offs(pOrigin,351.86,122.51,0.00),v40,z0,tPen\WObj:=wPaper;
    MoveL Offs(pOrigin,353.27,123.57,0.00),v40,z0,tPen\WObj:=wPaper;
    MoveL Offs(pOrigin,357.95,130.80,0.00),v40,z0,tPen\WObj:=wPaper;
    MoveL Offs(pOrigin,363.69,136.96,0.00),v40,z0,tPen\WObj:=wPaper;
    MoveL Offs(pOrigin,366.45,139.09,0.00),v40,z0,tPen\WObj:=wPaper;
    MoveL Offs(pOrigin,370.27,141.50,0.00),v40,z0,tPen\WObj:=wPaper;
    MoveL Offs(pOrigin,376.65,143.98,0.00),v40,fine,tPen\WObj:=wPaper;
    MoveL Offs(pOrigin,376.65,143.98,6.00),v60,z5,tPen\WObj:=wPaper;
    MoveL Offs(pOrigin,371.34,142.06,6.00),vTravel,z5,tPen\WObj:=wPaper;
    MoveL Offs(pOrigin,371.34,142.06,0.00),v60,z0,tPen\WObj:=wPaper;
    MoveL Offs(pOrigin,371.76,142.27,0.00),v40,z0,tPen\WObj:=wPaper;
    MoveL Offs(pOrigin,371.34,142.06,0.00),v40,fine,tPen\WObj:=wPaper;
    MoveL Offs(pOrigin,371.34,142.06,6.00),v60,z5,tPen\WObj:=wPaper;
    MoveL Offs(pOrigin,367.73,145.25,6.00),vTravel,z5,tPen\WObj:=wPaper;
    MoveL Offs(pOrigin,367.73,145.25,0.00),v60,z0,tPen\WObj:=wPaper;
    MoveL Offs(pOrigin,368.15,145.68,0.00),v40,z0,tPen\WObj:=wPaper;
    MoveL Offs(pOrigin,367.73,145.25,0.00),v40,fine,tPen\WObj:=wPaper;
    MoveL Offs(pOrigin,367.73,145.25,6.00),v60,z5,tPen\WObj:=wPaper;
    MoveL Offs(pOrigin,365.81,143.55,6.00),vTravel,z5,tPen\WObj:=wPaper;
    MoveL Offs(pOrigin,365.81,143.55,0.00),v60,z0,tPen\WObj:=wPaper;
    MoveL Offs(pOrigin,366.88,144.61,0.00),v40,z0,tPen\WObj:=wPaper;
    MoveL Offs(pOrigin,365.81,143.55,0.00),v40,fine,tPen\WObj:=wPaper;
    MoveL Offs(pOrigin,365.81,143.55,6.00),v60,z5,tPen\WObj:=wPaper;
    MoveL Offs(pOrigin,363.69,146.31,6.00),vTravel,z5,tPen\WObj:=wPaper;
    MoveL Offs(pOrigin,363.69,146.31,0.00),v60,z0,tPen\WObj:=wPaper;
    MoveL Offs(pOrigin,364.11,146.74,0.00),v40,z0,tPen\WObj:=wPaper;
    MoveL Offs(pOrigin,363.69,146.31,0.00),v40,fine,tPen\WObj:=wPaper;
    MoveL Offs(pOrigin,363.69,146.31,6.00),v60,z5,tPen\WObj:=wPaper;
    MoveL Offs(pOrigin,361.56,143.76,6.00),vTravel,z5,tPen\WObj:=wPaper;
    MoveL Offs(pOrigin,361.56,143.76,0.00),v60,z0,tPen\WObj:=wPaper;
    MoveL Offs(pOrigin,361.99,144.19,0.00),v40,z0,tPen\WObj:=wPaper;
    MoveL Offs(pOrigin,361.56,143.76,0.00),v40,fine,tPen\WObj:=wPaper;
    MoveL Offs(pOrigin,361.56,143.76,6.00),v60,z5,tPen\WObj:=wPaper;
    MoveL Offs(pOrigin,359.86,141.43,6.00),vTravel,z5,tPen\WObj:=wPaper;
    MoveL Offs(pOrigin,359.86,141.43,0.00),v60,z0,tPen\WObj:=wPaper;
    MoveL Offs(pOrigin,374.31,159.06,0.00),v40,z0,tPen\WObj:=wPaper;
    MoveL Offs(pOrigin,378.56,164.80,0.00),v40,z0,tPen\WObj:=wPaper;
    MoveL Offs(pOrigin,379.62,165.23,0.00),v40,fine,tPen\WObj:=wPaper;
    MoveL Offs(pOrigin,379.62,165.23,6.00),v60,z5,tPen\WObj:=wPaper;
    MoveL Offs(pOrigin,376.65,162.25,6.00),vTravel,z5,tPen\WObj:=wPaper;
    MoveL Offs(pOrigin,376.65,162.25,0.00),v60,z0,tPen\WObj:=wPaper;
    MoveL Offs(pOrigin,377.08,162.89,0.00),v40,z0,tPen\WObj:=wPaper;
    MoveL Offs(pOrigin,376.65,162.25,0.00),v40,fine,tPen\WObj:=wPaper;
    MoveL Offs(pOrigin,376.65,162.25,6.00),v60,z5,tPen\WObj:=wPaper;
    MoveL Offs(pOrigin,381.11,160.98,6.00),vTravel,z5,tPen\WObj:=wPaper;
    MoveL Offs(pOrigin,381.11,160.98,0.00),v60,z0,tPen\WObj:=wPaper;
    MoveL Offs(pOrigin,380.90,161.40,0.00),v40,z0,tPen\WObj:=wPaper;
    MoveL Offs(pOrigin,381.11,160.98,0.00),v40,fine,tPen\WObj:=wPaper;
    MoveL Offs(pOrigin,381.11,160.98,6.00),v60,z5,tPen\WObj:=wPaper;
    MoveL Offs(pOrigin,382.81,157.15,6.00),vTravel,z5,tPen\WObj:=wPaper;
    MoveL Offs(pOrigin,382.81,157.15,0.00),v60,z0,tPen\WObj:=wPaper;
    MoveL Offs(pOrigin,382.60,157.57,0.00),v40,z0,tPen\WObj:=wPaper;
    MoveL Offs(pOrigin,382.81,157.15,0.00),v40,z0,tPen\WObj:=wPaper;
    MoveL Offs(pOrigin,383.24,156.30,0.00),v40,z0,tPen\WObj:=wPaper;
    MoveL Offs(pOrigin,383.02,156.73,0.00),v40,z0,tPen\WObj:=wPaper;
    MoveL Offs(pOrigin,383.24,156.30,0.00),v40,fine,tPen\WObj:=wPaper;
    MoveL Offs(pOrigin,383.24,156.30,6.00),v60,z5,tPen\WObj:=wPaper;
    MoveL Offs(pOrigin,384.94,152.69,6.00),vTravel,z5,tPen\WObj:=wPaper;
    MoveL Offs(pOrigin,384.94,152.69,0.00),v60,z0,tPen\WObj:=wPaper;
    MoveL Offs(pOrigin,384.73,153.11,0.00),v40,z0,tPen\WObj:=wPaper;
    MoveL Offs(pOrigin,384.94,152.69,0.00),v40,z0,tPen\WObj:=wPaper;
    MoveL Offs(pOrigin,385.36,151.62,0.00),v40,z0,tPen\WObj:=wPaper;
    MoveL Offs(pOrigin,385.15,152.05,0.00),v40,z0,tPen\WObj:=wPaper;
    MoveL Offs(pOrigin,385.36,151.62,0.00),v40,fine,tPen\WObj:=wPaper;
    MoveL Offs(pOrigin,385.36,151.62,6.00),v60,z5,tPen\WObj:=wPaper;
    MoveL Offs(pOrigin,374.95,150.56,6.00),vTravel,z5,tPen\WObj:=wPaper;
    MoveL Offs(pOrigin,374.95,150.56,0.00),v60,z0,tPen\WObj:=wPaper;
    MoveL Offs(pOrigin,372.40,149.07,0.00),v40,z0,tPen\WObj:=wPaper;
    MoveL Offs(pOrigin,367.94,145.68,0.00),v40,z0,tPen\WObj:=wPaper;
    MoveL Offs(pOrigin,362.84,141.00,0.00),v40,z0,tPen\WObj:=wPaper;
    MoveL Offs(pOrigin,356.67,133.77,0.00),v40,z0,tPen\WObj:=wPaper;
    MoveL Offs(pOrigin,353.91,129.52,0.00),v40,z0,tPen\WObj:=wPaper;
    MoveL Offs(pOrigin,352.64,128.68,0.00),v40,z0,tPen\WObj:=wPaper;
    MoveL Offs(pOrigin,352.64,128.68,0.00),v40,z0,tPen\WObj:=wPaper;
    MoveL Offs(pOrigin,352.64,130.38,0.00),v40,z0,tPen\WObj:=wPaper;
    MoveL Offs(pOrigin,355.61,143.76,0.00),v40,z0,tPen\WObj:=wPaper;
    MoveL Offs(pOrigin,362.84,170.96,0.00),v40,z0,tPen\WObj:=wPaper;
    MoveL Offs(pOrigin,367.02,183.29,0.00),v40,z0,tPen\WObj:=wPaper;
    MoveL Offs(pOrigin,368.50,186.48,0.00),v40,z0,tPen\WObj:=wPaper;
    MoveL Offs(pOrigin,370.70,189.88,0.00),v40,z0,tPen\WObj:=wPaper;
    MoveL Offs(pOrigin,370.70,189.88,0.00),v40,z0,tPen\WObj:=wPaper;
    MoveL Offs(pOrigin,373.04,189.88,0.00),v40,z0,tPen\WObj:=wPaper;
    MoveL Offs(pOrigin,373.04,189.88,0.00),v40,z0,tPen\WObj:=wPaper;
    MoveL Offs(pOrigin,376.23,206.24,0.00),v40,z0,tPen\WObj:=wPaper;
    MoveL Offs(pOrigin,376.65,213.04,0.00),v40,z0,tPen\WObj:=wPaper;
    MoveL Offs(pOrigin,376.65,213.04,0.00),v40,z0,tPen\WObj:=wPaper;
    MoveL Offs(pOrigin,377.08,215.59,0.00),v40,z0,tPen\WObj:=wPaper;
    MoveL Offs(pOrigin,377.08,219.84,0.00),v40,z0,tPen\WObj:=wPaper;
    MoveL Offs(pOrigin,376.44,225.57,0.00),v40,z0,tPen\WObj:=wPaper;
  ENDPROC

  PROC DrawPart17()
    MoveL Offs(pOrigin,375.02,230.68,0.00),v40,z0,tPen\WObj:=wPaper;
    MoveL Offs(pOrigin,373.25,233.86,0.00),v40,z0,tPen\WObj:=wPaper;
    MoveL Offs(pOrigin,370.91,236.13,0.00),v40,z0,tPen\WObj:=wPaper;
    MoveL Offs(pOrigin,367.30,237.97,0.00),v40,z0,tPen\WObj:=wPaper;
    MoveL Offs(pOrigin,363.05,239.18,0.00),v40,z0,tPen\WObj:=wPaper;
    MoveL Offs(pOrigin,358.38,239.60,0.00),v40,fine,tPen\WObj:=wPaper;
    MoveL Offs(pOrigin,358.38,239.60,6.00),v60,z5,tPen\WObj:=wPaper;
    MoveL Offs(pOrigin,364.75,233.65,6.00),vTravel,z5,tPen\WObj:=wPaper;
    MoveL Offs(pOrigin,364.75,233.65,0.00),v60,z0,tPen\WObj:=wPaper;
    MoveL Offs(pOrigin,365.17,233.44,0.00),v40,z0,tPen\WObj:=wPaper;
    MoveL Offs(pOrigin,364.75,233.65,0.00),v40,fine,tPen\WObj:=wPaper;
    MoveL Offs(pOrigin,364.75,233.65,6.00),v60,z5,tPen\WObj:=wPaper;
    MoveL Offs(pOrigin,370.49,229.40,6.00),vTravel,z5,tPen\WObj:=wPaper;
    MoveL Offs(pOrigin,370.49,229.40,0.00),v60,z0,tPen\WObj:=wPaper;
    MoveL Offs(pOrigin,370.27,229.82,0.00),v40,z0,tPen\WObj:=wPaper;
    MoveL Offs(pOrigin,370.49,229.40,0.00),v40,fine,tPen\WObj:=wPaper;
    MoveL Offs(pOrigin,370.49,229.40,6.00),v60,z5,tPen\WObj:=wPaper;
    MoveL Offs(pOrigin,371.34,228.34,6.00),vTravel,z5,tPen\WObj:=wPaper;
    MoveL Offs(pOrigin,371.34,228.34,0.00),v60,z0,tPen\WObj:=wPaper;
    MoveL Offs(pOrigin,371.12,228.76,0.00),v40,z0,tPen\WObj:=wPaper;
    MoveL Offs(pOrigin,371.34,228.34,0.00),v40,fine,tPen\WObj:=wPaper;
    MoveL Offs(pOrigin,371.34,228.34,6.00),v60,z5,tPen\WObj:=wPaper;
    MoveL Offs(pOrigin,371.98,227.27,6.00),vTravel,z5,tPen\WObj:=wPaper;
    MoveL Offs(pOrigin,371.98,227.27,0.00),v60,z0,tPen\WObj:=wPaper;
    MoveL Offs(pOrigin,371.76,227.70,0.00),v40,z0,tPen\WObj:=wPaper;
    MoveL Offs(pOrigin,371.98,227.27,0.00),v40,z0,tPen\WObj:=wPaper;
    MoveL Offs(pOrigin,372.40,226.43,0.00),v40,z0,tPen\WObj:=wPaper;
    MoveL Offs(pOrigin,372.19,226.85,0.00),v40,z0,tPen\WObj:=wPaper;
    MoveL Offs(pOrigin,372.40,226.43,0.00),v40,z0,tPen\WObj:=wPaper;
    MoveL Offs(pOrigin,372.83,225.57,0.00),v40,z0,tPen\WObj:=wPaper;
    MoveL Offs(pOrigin,372.61,226.00,0.00),v40,z0,tPen\WObj:=wPaper;
    MoveL Offs(pOrigin,372.83,225.57,0.00),v40,z0,tPen\WObj:=wPaper;
    MoveL Offs(pOrigin,373.25,224.73,0.00),v40,z0,tPen\WObj:=wPaper;
    MoveL Offs(pOrigin,373.04,225.15,0.00),v40,z0,tPen\WObj:=wPaper;
    MoveL Offs(pOrigin,373.25,224.73,0.00),v40,fine,tPen\WObj:=wPaper;
    MoveL Offs(pOrigin,373.25,224.73,6.00),v60,z5,tPen\WObj:=wPaper;
    MoveL Offs(pOrigin,377.50,233.23,6.00),vTravel,z5,tPen\WObj:=wPaper;
    MoveL Offs(pOrigin,377.50,233.23,0.00),v60,z0,tPen\WObj:=wPaper;
    MoveL Offs(pOrigin,377.29,233.65,0.00),v40,z0,tPen\WObj:=wPaper;
    MoveL Offs(pOrigin,377.50,233.23,0.00),v40,fine,tPen\WObj:=wPaper;
    MoveL Offs(pOrigin,377.50,233.23,6.00),v60,z5,tPen\WObj:=wPaper;
    MoveL Offs(pOrigin,377.29,234.50,6.00),vTravel,z5,tPen\WObj:=wPaper;
    MoveL Offs(pOrigin,377.29,234.50,0.00),v60,z0,tPen\WObj:=wPaper;
    MoveL Offs(pOrigin,377.36,235.14,0.00),v40,z0,tPen\WObj:=wPaper;
    MoveL Offs(pOrigin,375.80,236.98,0.00),v40,z0,tPen\WObj:=wPaper;
    MoveL Offs(pOrigin,372.61,239.03,0.00),v40,z0,tPen\WObj:=wPaper;
    MoveL Offs(pOrigin,366.45,241.09,0.00),v40,z0,tPen\WObj:=wPaper;
    MoveL Offs(pOrigin,358.16,242.57,0.00),v40,z0,tPen\WObj:=wPaper;
    MoveL Offs(pOrigin,345.20,244.06,0.00),v40,z0,tPen\WObj:=wPaper;
    MoveL Offs(pOrigin,327.99,245.34,0.00),v40,z0,tPen\WObj:=wPaper;
    MoveL Offs(pOrigin,317.15,245.76,0.00),v40,z0,tPen\WObj:=wPaper;
    MoveL Offs(pOrigin,298.66,245.76,0.00),v40,z0,tPen\WObj:=wPaper;
    MoveL Offs(pOrigin,298.66,245.76,0.00),v40,z0,tPen\WObj:=wPaper;
    MoveL Offs(pOrigin,298.24,245.12,0.00),v40,z0,tPen\WObj:=wPaper;
    MoveL Offs(pOrigin,297.25,240.45,0.00),v40,z0,tPen\WObj:=wPaper;
    MoveL Offs(pOrigin,295.48,238.61,0.00),v40,z0,tPen\WObj:=wPaper;
    MoveL Offs(pOrigin,294.62,238.32,0.00),v40,z0,tPen\WObj:=wPaper;
    MoveL Offs(pOrigin,291.44,238.54,0.00),v40,z0,tPen\WObj:=wPaper;
    MoveL Offs(pOrigin,291.44,238.54,0.00),v40,z0,tPen\WObj:=wPaper;
    MoveL Offs(pOrigin,290.59,247.68,0.00),v40,fine,tPen\WObj:=wPaper;
    MoveL Offs(pOrigin,290.59,247.68,6.00),v60,z5,tPen\WObj:=wPaper;
    MoveL Offs(pOrigin,290.80,250.01,6.00),vTravel,z5,tPen\WObj:=wPaper;
    MoveL Offs(pOrigin,290.80,250.01,0.00),v60,z0,tPen\WObj:=wPaper;
    MoveL Offs(pOrigin,291.86,252.14,0.00),v40,z0,tPen\WObj:=wPaper;
    MoveL Offs(pOrigin,291.86,252.14,0.00),v40,z0,tPen\WObj:=wPaper;
    MoveL Offs(pOrigin,292.50,255.11,0.00),v40,z0,tPen\WObj:=wPaper;
    MoveL Offs(pOrigin,291.72,257.66,0.00),v40,z0,tPen\WObj:=wPaper;
    MoveL Offs(pOrigin,289.74,260.64,0.00),v40,z0,tPen\WObj:=wPaper;
    MoveL Offs(pOrigin,290.80,260.85,0.00),v40,z0,tPen\WObj:=wPaper;
    MoveL Offs(pOrigin,292.92,258.09,0.00),v40,fine,tPen\WObj:=wPaper;
    MoveL Offs(pOrigin,292.92,258.09,6.00),v60,z5,tPen\WObj:=wPaper;
    MoveL Offs(pOrigin,291.65,257.45,6.00),vTravel,z5,tPen\WObj:=wPaper;
    MoveL Offs(pOrigin,291.65,257.45,0.00),v60,z0,tPen\WObj:=wPaper;
    MoveL Offs(pOrigin,291.44,257.88,0.00),v40,z0,tPen\WObj:=wPaper;
    MoveL Offs(pOrigin,291.65,257.45,0.00),v40,fine,tPen\WObj:=wPaper;
    MoveL Offs(pOrigin,291.65,257.45,6.00),v60,z5,tPen\WObj:=wPaper;
    MoveL Offs(pOrigin,294.84,256.39,6.00),vTravel,z5,tPen\WObj:=wPaper;
    MoveL Offs(pOrigin,294.84,256.39,0.00),v60,z0,tPen\WObj:=wPaper;
    MoveL Offs(pOrigin,293.77,253.41,0.00),v40,z0,tPen\WObj:=wPaper;
    MoveL Offs(pOrigin,292.92,252.56,0.00),v40,z0,tPen\WObj:=wPaper;
    MoveL Offs(pOrigin,291.86,252.14,0.00),v40,fine,tPen\WObj:=wPaper;
    MoveL Offs(pOrigin,291.86,252.14,6.00),v60,z5,tPen\WObj:=wPaper;
    MoveL Offs(pOrigin,294.20,253.84,6.00),vTravel,z5,tPen\WObj:=wPaper;
    MoveL Offs(pOrigin,294.20,253.84,0.00),v60,z0,tPen\WObj:=wPaper;
    MoveL Offs(pOrigin,294.41,254.26,0.00),v40,z0,tPen\WObj:=wPaper;
    MoveL Offs(pOrigin,294.20,253.84,0.00),v40,fine,tPen\WObj:=wPaper;
    MoveL Offs(pOrigin,294.20,253.84,6.00),v60,z5,tPen\WObj:=wPaper;
    MoveL Offs(pOrigin,295.26,249.80,6.00),vTravel,z5,tPen\WObj:=wPaper;
    MoveL Offs(pOrigin,295.26,249.80,0.00),v60,z0,tPen\WObj:=wPaper;
    MoveL Offs(pOrigin,297.03,252.56,0.00),v40,z0,tPen\WObj:=wPaper;
    MoveL Offs(pOrigin,298.24,256.81,0.00),v40,z0,tPen\WObj:=wPaper;
    MoveL Offs(pOrigin,298.24,258.09,0.00),v40,z0,tPen\WObj:=wPaper;
    MoveL Offs(pOrigin,299.09,259.58,0.00),v40,z0,tPen\WObj:=wPaper;
    MoveL Offs(pOrigin,299.94,264.89,0.00),v40,z0,tPen\WObj:=wPaper;
    MoveL Offs(pOrigin,299.73,266.38,0.00),v40,z0,tPen\WObj:=wPaper;
    MoveL Offs(pOrigin,298.80,269.14,0.00),v40,z0,tPen\WObj:=wPaper;
    MoveL Offs(pOrigin,297.81,270.55,0.00),v40,z0,tPen\WObj:=wPaper;
    MoveL Offs(pOrigin,296.33,271.26,0.00),v40,z0,tPen\WObj:=wPaper;
    MoveL Offs(pOrigin,295.05,270.91,0.00),v40,z0,tPen\WObj:=wPaper;
    MoveL Offs(pOrigin,293.56,269.77,0.00),v40,z0,tPen\WObj:=wPaper;
    MoveL Offs(pOrigin,291.15,266.16,0.00),v40,z0,tPen\WObj:=wPaper;
    MoveL Offs(pOrigin,290.16,263.40,0.00),v40,z0,tPen\WObj:=wPaper;
    MoveL Offs(pOrigin,289.95,261.70,0.00),v40,z0,tPen\WObj:=wPaper;
    MoveL Offs(pOrigin,289.95,261.70,0.00),v40,z0,tPen\WObj:=wPaper;
    MoveL Offs(pOrigin,289.88,261.06,0.00),v40,z0,tPen\WObj:=wPaper;
    MoveL Offs(pOrigin,289.31,260.71,0.00),v40,z0,tPen\WObj:=wPaper;
    MoveL Offs(pOrigin,287.83,261.91,0.00),v40,z0,tPen\WObj:=wPaper;
    MoveL Offs(pOrigin,287.83,261.91,0.00),v40,z0,tPen\WObj:=wPaper;
    MoveL Offs(pOrigin,287.61,264.04,0.00),v40,z0,tPen\WObj:=wPaper;
    MoveL Offs(pOrigin,288.18,264.89,0.00),v40,z0,tPen\WObj:=wPaper;
    MoveL Offs(pOrigin,288.25,265.74,0.00),v40,z0,tPen\WObj:=wPaper;
    MoveL Offs(pOrigin,288.25,265.74,0.00),v40,z0,tPen\WObj:=wPaper;
    MoveL Offs(pOrigin,288.04,266.80,0.00),v40,z0,tPen\WObj:=wPaper;
    MoveL Offs(pOrigin,288.04,267.23,0.00),v40,z0,tPen\WObj:=wPaper;
    MoveL Offs(pOrigin,287.83,266.80,0.00),v40,z0,tPen\WObj:=wPaper;
    MoveL Offs(pOrigin,285.91,266.80,0.00),v40,z0,tPen\WObj:=wPaper;
    MoveL Offs(pOrigin,285.91,266.80,0.00),v40,z0,tPen\WObj:=wPaper;
    MoveL Offs(pOrigin,286.34,265.10,0.00),v40,z0,tPen\WObj:=wPaper;
    MoveL Offs(pOrigin,287.61,264.46,0.00),v40,fine,tPen\WObj:=wPaper;
    MoveL Offs(pOrigin,287.61,264.46,6.00),v60,z5,tPen\WObj:=wPaper;
  ENDPROC

  PROC DrawPart18()
    MoveL Offs(pOrigin,287.83,261.91,6.00),vTravel,z5,tPen\WObj:=wPaper;
    MoveL Offs(pOrigin,287.83,261.91,0.00),v60,z0,tPen\WObj:=wPaper;
    MoveL Offs(pOrigin,287.61,261.49,0.00),v40,z0,tPen\WObj:=wPaper;
    MoveL Offs(pOrigin,287.83,258.94,0.00),v40,fine,tPen\WObj:=wPaper;
    MoveL Offs(pOrigin,287.83,258.94,6.00),v60,z5,tPen\WObj:=wPaper;
    MoveL Offs(pOrigin,289.95,261.70,6.00),vTravel,z5,tPen\WObj:=wPaper;
    MoveL Offs(pOrigin,289.95,261.70,0.00),v60,z0,tPen\WObj:=wPaper;
    MoveL Offs(pOrigin,291.65,261.27,0.00),v40,fine,tPen\WObj:=wPaper;
    MoveL Offs(pOrigin,291.65,261.27,6.00),v60,z5,tPen\WObj:=wPaper;
    MoveL Offs(pOrigin,291.23,265.95,6.00),vTravel,z5,tPen\WObj:=wPaper;
    MoveL Offs(pOrigin,291.23,265.95,0.00),v60,z0,tPen\WObj:=wPaper;
    MoveL Offs(pOrigin,291.44,266.38,0.00),v40,z0,tPen\WObj:=wPaper;
    MoveL Offs(pOrigin,291.23,265.95,0.00),v40,fine,tPen\WObj:=wPaper;
    MoveL Offs(pOrigin,291.23,265.95,6.00),v60,z5,tPen\WObj:=wPaper;
    MoveL Offs(pOrigin,287.83,268.08,6.00),vTravel,z5,tPen\WObj:=wPaper;
    MoveL Offs(pOrigin,287.83,268.08,0.00),v60,z0,tPen\WObj:=wPaper;
    MoveL Offs(pOrigin,288.04,270.62,0.00),v40,z0,tPen\WObj:=wPaper;
    MoveL Offs(pOrigin,288.04,270.62,0.00),v40,z0,tPen\WObj:=wPaper;
    MoveL Offs(pOrigin,286.76,270.84,0.00),v40,z0,tPen\WObj:=wPaper;
    MoveL Offs(pOrigin,285.06,270.55,0.00),v40,z0,tPen\WObj:=wPaper;
    MoveL Offs(pOrigin,284.85,270.20,0.00),v40,z0,tPen\WObj:=wPaper;
    MoveL Offs(pOrigin,285.06,268.92,0.00),v40,z0,tPen\WObj:=wPaper;
    MoveL Offs(pOrigin,285.49,268.29,0.00),v40,z0,tPen\WObj:=wPaper;
    MoveL Offs(pOrigin,285.49,268.29,0.00),v40,z0,tPen\WObj:=wPaper;
    MoveL Offs(pOrigin,285.91,266.80,0.00),v40,fine,tPen\WObj:=wPaper;
    MoveL Offs(pOrigin,285.91,266.80,6.00),v60,z5,tPen\WObj:=wPaper;
    MoveL Offs(pOrigin,285.49,268.29,6.00),vTravel,z5,tPen\WObj:=wPaper;
    MoveL Offs(pOrigin,285.49,268.29,0.00),v60,z0,tPen\WObj:=wPaper;
    MoveL Offs(pOrigin,287.83,268.08,0.00),v40,fine,tPen\WObj:=wPaper;
    MoveL Offs(pOrigin,287.83,268.08,6.00),v60,z5,tPen\WObj:=wPaper;
    MoveL Offs(pOrigin,288.89,270.84,6.00),vTravel,z5,tPen\WObj:=wPaper;
    MoveL Offs(pOrigin,288.89,270.84,0.00),v60,z0,tPen\WObj:=wPaper;
    MoveL Offs(pOrigin,289.31,272.25,0.00),v40,z0,tPen\WObj:=wPaper;
    MoveL Offs(pOrigin,291.01,272.61,0.00),v40,z0,tPen\WObj:=wPaper;
    MoveL Offs(pOrigin,293.14,274.02,0.00),v40,z0,tPen\WObj:=wPaper;
    MoveL Offs(pOrigin,294.20,275.73,0.00),v40,z0,tPen\WObj:=wPaper;
    MoveL Offs(pOrigin,294.62,275.73,0.00),v40,z0,tPen\WObj:=wPaper;
    MoveL Offs(pOrigin,295.48,275.09,0.00),v40,z0,tPen\WObj:=wPaper;
    MoveL Offs(pOrigin,297.81,275.30,0.00),v40,z0,tPen\WObj:=wPaper;
    MoveL Offs(pOrigin,297.81,275.30,0.00),v40,z0,tPen\WObj:=wPaper;
    MoveL Offs(pOrigin,298.66,275.94,0.00),v40,z0,tPen\WObj:=wPaper;
    MoveL Offs(pOrigin,298.66,277.64,0.00),v40,z0,tPen\WObj:=wPaper;
    MoveL Offs(pOrigin,298.02,278.91,0.00),v40,z0,tPen\WObj:=wPaper;
    MoveL Offs(pOrigin,297.60,278.91,0.00),v40,z0,tPen\WObj:=wPaper;
    MoveL Offs(pOrigin,298.24,279.98,0.00),v40,z0,tPen\WObj:=wPaper;
    MoveL Offs(pOrigin,298.24,281.67,0.00),v40,z0,tPen\WObj:=wPaper;
    MoveL Offs(pOrigin,298.24,281.67,0.00),v40,z0,tPen\WObj:=wPaper;
    MoveL Offs(pOrigin,297.39,282.10,0.00),v40,z0,tPen\WObj:=wPaper;
    MoveL Offs(pOrigin,297.39,282.10,0.00),v40,z0,tPen\WObj:=wPaper;
    MoveL Offs(pOrigin,296.54,281.46,0.00),v40,z0,tPen\WObj:=wPaper;
    MoveL Offs(pOrigin,296.54,281.46,0.00),v40,z0,tPen\WObj:=wPaper;
    MoveL Offs(pOrigin,295.83,279.55,0.00),v40,z0,tPen\WObj:=wPaper;
    MoveL Offs(pOrigin,294.41,278.06,0.00),v40,z0,tPen\WObj:=wPaper;
    MoveL Offs(pOrigin,294.41,278.06,0.00),v40,z0,tPen\WObj:=wPaper;
    MoveL Offs(pOrigin,293.35,278.27,0.00),v40,z0,tPen\WObj:=wPaper;
    MoveL Offs(pOrigin,291.86,277.85,0.00),v40,z0,tPen\WObj:=wPaper;
    MoveL Offs(pOrigin,289.74,277.85,0.00),v40,z0,tPen\WObj:=wPaper;
    MoveL Offs(pOrigin,289.31,277.42,0.00),v40,z0,tPen\WObj:=wPaper;
    MoveL Offs(pOrigin,289.31,277.42,0.00),v40,z0,tPen\WObj:=wPaper;
    MoveL Offs(pOrigin,289.31,277.00,0.00),v40,z0,tPen\WObj:=wPaper;
    MoveL Offs(pOrigin,290.16,276.79,0.00),v40,z0,tPen\WObj:=wPaper;
    MoveL Offs(pOrigin,290.80,276.15,0.00),v40,z0,tPen\WObj:=wPaper;
    MoveL Offs(pOrigin,290.80,276.15,0.00),v40,z0,tPen\WObj:=wPaper;
    MoveL Offs(pOrigin,294.41,275.87,0.00),v40,z0,tPen\WObj:=wPaper;
    MoveL Offs(pOrigin,294.84,277.21,0.00),v40,z0,tPen\WObj:=wPaper;
    MoveL Offs(pOrigin,294.84,277.21,0.00),v40,z0,tPen\WObj:=wPaper;
    MoveL Offs(pOrigin,295.26,277.42,0.00),v40,z0,tPen\WObj:=wPaper;
    MoveL Offs(pOrigin,295.05,277.64,0.00),v40,z0,tPen\WObj:=wPaper;
    MoveL Offs(pOrigin,294.84,277.42,0.00),v40,z0,tPen\WObj:=wPaper;
    MoveL Offs(pOrigin,295.26,277.21,0.00),v40,z0,tPen\WObj:=wPaper;
    MoveL Offs(pOrigin,296.54,277.00,0.00),v40,z0,tPen\WObj:=wPaper;
    MoveL Offs(pOrigin,296.54,277.00,0.00),v40,z0,tPen\WObj:=wPaper;
    MoveL Offs(pOrigin,296.75,277.85,0.00),v40,z0,tPen\WObj:=wPaper;
    MoveL Offs(pOrigin,297.60,278.91,0.00),v40,z0,tPen\WObj:=wPaper;
    MoveL Offs(pOrigin,297.60,278.91,0.00),v40,z0,tPen\WObj:=wPaper;
    MoveL Offs(pOrigin,296.96,278.27,0.00),v40,z0,tPen\WObj:=wPaper;
    MoveL Offs(pOrigin,297.60,278.91,0.00),v40,z0,tPen\WObj:=wPaper;
    MoveL Offs(pOrigin,295.69,279.12,0.00),v40,fine,tPen\WObj:=wPaper;
    MoveL Offs(pOrigin,295.69,279.12,6.00),v60,z5,tPen\WObj:=wPaper;
    MoveL Offs(pOrigin,296.54,277.00,6.00),vTravel,z5,tPen\WObj:=wPaper;
    MoveL Offs(pOrigin,296.54,277.00,0.00),v60,z0,tPen\WObj:=wPaper;
    MoveL Offs(pOrigin,297.17,276.79,0.00),v40,z0,tPen\WObj:=wPaper;
    MoveL Offs(pOrigin,297.17,276.36,0.00),v40,z0,tPen\WObj:=wPaper;
    MoveL Offs(pOrigin,297.81,275.73,0.00),v40,z0,tPen\WObj:=wPaper;
    MoveL Offs(pOrigin,298.66,275.51,0.00),v40,z0,tPen\WObj:=wPaper;
    MoveL Offs(pOrigin,299.37,273.60,0.00),v40,z0,tPen\WObj:=wPaper;
    MoveL Offs(pOrigin,301.50,269.99,0.00),v40,z0,tPen\WObj:=wPaper;
    MoveL Offs(pOrigin,302.49,266.59,0.00),v40,z0,tPen\WObj:=wPaper;
    MoveL Offs(pOrigin,302.70,264.04,0.00),v40,z0,tPen\WObj:=wPaper;
    MoveL Offs(pOrigin,302.27,261.27,0.00),v40,z0,tPen\WObj:=wPaper;
    MoveL Offs(pOrigin,299.09,249.38,0.00),v40,z0,tPen\WObj:=wPaper;
    MoveL Offs(pOrigin,298.66,245.76,0.00),v40,z0,tPen\WObj:=wPaper;
    MoveL Offs(pOrigin,298.45,245.34,0.00),v40,z0,tPen\WObj:=wPaper;
    MoveL Offs(pOrigin,298.66,245.76,0.00),v40,z0,tPen\WObj:=wPaper;
    MoveL Offs(pOrigin,298.45,245.34,0.00),v40,fine,tPen\WObj:=wPaper;
    MoveL Offs(pOrigin,298.45,245.34,6.00),v60,z5,tPen\WObj:=wPaper;
    MoveL Offs(pOrigin,297.17,240.02,6.00),vTravel,z5,tPen\WObj:=wPaper;
    MoveL Offs(pOrigin,297.17,240.02,0.00),v60,z0,tPen\WObj:=wPaper;
    MoveL Offs(pOrigin,297.81,239.60,0.00),v40,z0,tPen\WObj:=wPaper;
    MoveL Offs(pOrigin,312.26,239.81,0.00),v40,z0,tPen\WObj:=wPaper;
    MoveL Offs(pOrigin,323.10,239.39,0.00),v40,z0,tPen\WObj:=wPaper;
    MoveL Offs(pOrigin,336.70,238.32,0.00),v40,z0,tPen\WObj:=wPaper;
    MoveL Offs(pOrigin,352.00,236.62,0.00),v40,z0,tPen\WObj:=wPaper;
    MoveL Offs(pOrigin,358.16,235.56,0.00),v40,z0,tPen\WObj:=wPaper;
    MoveL Offs(pOrigin,363.26,234.15,0.00),v40,z0,tPen\WObj:=wPaper;
    MoveL Offs(pOrigin,366.66,232.66,0.00),v40,z0,tPen\WObj:=wPaper;
    MoveL Offs(pOrigin,368.36,231.52,0.00),v40,z0,tPen\WObj:=wPaper;
    MoveL Offs(pOrigin,370.63,229.40,0.00),v40,z0,tPen\WObj:=wPaper;
    MoveL Offs(pOrigin,372.05,227.49,0.00),v40,z0,tPen\WObj:=wPaper;
    MoveL Offs(pOrigin,373.32,224.94,0.00),v40,z0,tPen\WObj:=wPaper;
    MoveL Offs(pOrigin,374.52,221.32,0.00),v40,z0,tPen\WObj:=wPaper;
    MoveL Offs(pOrigin,375.38,217.29,0.00),v40,z0,tPen\WObj:=wPaper;
    MoveL Offs(pOrigin,375.59,214.10,0.00),v40,z0,tPen\WObj:=wPaper;
    MoveL Offs(pOrigin,376.65,213.04,0.00),v40,fine,tPen\WObj:=wPaper;
    MoveL Offs(pOrigin,376.65,213.04,6.00),v60,z5,tPen\WObj:=wPaper;
    MoveL Offs(pOrigin,372.19,234.93,6.00),vTravel,z5,tPen\WObj:=wPaper;
    MoveL Offs(pOrigin,372.19,234.93,0.00),v60,z0,tPen\WObj:=wPaper;
    MoveL Offs(pOrigin,371.98,235.35,0.00),v40,z0,tPen\WObj:=wPaper;
    MoveL Offs(pOrigin,372.19,234.93,0.00),v40,fine,tPen\WObj:=wPaper;
    MoveL Offs(pOrigin,372.19,234.93,6.00),v60,z5,tPen\WObj:=wPaper;
  ENDPROC

  PROC DrawPart19()
    MoveL Offs(pOrigin,372.61,239.18,6.00),vTravel,z5,tPen\WObj:=wPaper;
    MoveL Offs(pOrigin,372.61,239.18,0.00),v60,z0,tPen\WObj:=wPaper;
    MoveL Offs(pOrigin,373.04,238.96,0.00),v40,z0,tPen\WObj:=wPaper;
    MoveL Offs(pOrigin,372.61,239.18,0.00),v40,z0,tPen\WObj:=wPaper;
    MoveL Offs(pOrigin,371.55,239.60,0.00),v40,z0,tPen\WObj:=wPaper;
    MoveL Offs(pOrigin,371.98,239.39,0.00),v40,z0,tPen\WObj:=wPaper;
    MoveL Offs(pOrigin,371.55,239.60,0.00),v40,fine,tPen\WObj:=wPaper;
    MoveL Offs(pOrigin,371.55,239.60,6.00),v60,z5,tPen\WObj:=wPaper;
    MoveL Offs(pOrigin,376.65,235.99,6.00),vTravel,z5,tPen\WObj:=wPaper;
    MoveL Offs(pOrigin,376.65,235.99,0.00),v60,z0,tPen\WObj:=wPaper;
    MoveL Offs(pOrigin,376.44,236.41,0.00),v40,z0,tPen\WObj:=wPaper;
    MoveL Offs(pOrigin,376.65,235.99,0.00),v40,fine,tPen\WObj:=wPaper;
    MoveL Offs(pOrigin,376.65,235.99,6.00),v60,z5,tPen\WObj:=wPaper;
    MoveL Offs(pOrigin,373.04,189.88,6.00),vTravel,z5,tPen\WObj:=wPaper;
    MoveL Offs(pOrigin,373.04,189.88,0.00),v60,z0,tPen\WObj:=wPaper;
    MoveL Offs(pOrigin,375.52,188.18,0.00),v40,z0,tPen\WObj:=wPaper;
    MoveL Offs(pOrigin,376.44,186.48,0.00),v40,z0,tPen\WObj:=wPaper;
    MoveL Offs(pOrigin,372.33,178.82,0.00),v40,z0,tPen\WObj:=wPaper;
    MoveL Offs(pOrigin,370.27,173.09,0.00),v40,fine,tPen\WObj:=wPaper;
    MoveL Offs(pOrigin,370.27,173.09,6.00),v60,z5,tPen\WObj:=wPaper;
    MoveL Offs(pOrigin,375.80,172.88,6.00),vTravel,z5,tPen\WObj:=wPaper;
    MoveL Offs(pOrigin,375.80,172.88,0.00),v60,z0,tPen\WObj:=wPaper;
    MoveL Offs(pOrigin,376.01,173.30,0.00),v40,z0,tPen\WObj:=wPaper;
    MoveL Offs(pOrigin,375.80,172.88,0.00),v40,z0,tPen\WObj:=wPaper;
    MoveL Offs(pOrigin,376.01,173.30,0.00),v40,z0,tPen\WObj:=wPaper;
    MoveL Offs(pOrigin,367.44,159.49,0.00),v40,z0,tPen\WObj:=wPaper;
    MoveL Offs(pOrigin,363.05,151.20,0.00),v40,fine,tPen\WObj:=wPaper;
    MoveL Offs(pOrigin,363.05,151.20,6.00),v60,z5,tPen\WObj:=wPaper;
    MoveL Offs(pOrigin,364.11,153.54,6.00),vTravel,z5,tPen\WObj:=wPaper;
    MoveL Offs(pOrigin,364.11,153.54,0.00),v60,z0,tPen\WObj:=wPaper;
    MoveL Offs(pOrigin,364.33,153.96,0.00),v40,z0,tPen\WObj:=wPaper;
    MoveL Offs(pOrigin,364.11,153.54,0.00),v40,fine,tPen\WObj:=wPaper;
    MoveL Offs(pOrigin,364.11,153.54,6.00),v60,z5,tPen\WObj:=wPaper;
    MoveL Offs(pOrigin,365.17,155.45,6.00),vTravel,z5,tPen\WObj:=wPaper;
    MoveL Offs(pOrigin,365.17,155.45,0.00),v60,z0,tPen\WObj:=wPaper;
    MoveL Offs(pOrigin,365.39,155.88,0.00),v40,z0,tPen\WObj:=wPaper;
    MoveL Offs(pOrigin,365.17,155.45,0.00),v40,z0,tPen\WObj:=wPaper;
    MoveL Offs(pOrigin,365.60,156.30,0.00),v40,z0,tPen\WObj:=wPaper;
    MoveL Offs(pOrigin,365.81,156.73,0.00),v40,z0,tPen\WObj:=wPaper;
    MoveL Offs(pOrigin,365.60,156.30,0.00),v40,fine,tPen\WObj:=wPaper;
    MoveL Offs(pOrigin,365.60,156.30,6.00),v60,z5,tPen\WObj:=wPaper;
    MoveL Offs(pOrigin,367.30,150.77,6.00),vTravel,z5,tPen\WObj:=wPaper;
    MoveL Offs(pOrigin,367.30,150.77,0.00),v60,z0,tPen\WObj:=wPaper;
    MoveL Offs(pOrigin,367.73,151.20,0.00),v40,z0,tPen\WObj:=wPaper;
    MoveL Offs(pOrigin,367.30,150.77,0.00),v40,fine,tPen\WObj:=wPaper;
    MoveL Offs(pOrigin,367.30,150.77,6.00),v60,z5,tPen\WObj:=wPaper;
    MoveL Offs(pOrigin,361.99,139.94,6.00),vTravel,z5,tPen\WObj:=wPaper;
    MoveL Offs(pOrigin,361.99,139.94,0.00),v60,z0,tPen\WObj:=wPaper;
    MoveL Offs(pOrigin,362.41,140.36,0.00),v40,z0,tPen\WObj:=wPaper;
    MoveL Offs(pOrigin,361.99,139.94,0.00),v40,fine,tPen\WObj:=wPaper;
    MoveL Offs(pOrigin,361.99,139.94,6.00),v60,z5,tPen\WObj:=wPaper;
    MoveL Offs(pOrigin,361.14,134.62,6.00),vTravel,z5,tPen\WObj:=wPaper;
    MoveL Offs(pOrigin,361.14,134.62,0.00),v60,z0,tPen\WObj:=wPaper;
    MoveL Offs(pOrigin,362.20,135.69,0.00),v40,z0,tPen\WObj:=wPaper;
    MoveL Offs(pOrigin,361.14,134.62,0.00),v40,fine,tPen\WObj:=wPaper;
    MoveL Offs(pOrigin,361.14,134.62,6.00),v60,z5,tPen\WObj:=wPaper;
    MoveL Offs(pOrigin,355.83,128.04,6.00),vTravel,z5,tPen\WObj:=wPaper;
    MoveL Offs(pOrigin,355.83,128.04,0.00),v60,z0,tPen\WObj:=wPaper;
    MoveL Offs(pOrigin,356.25,128.68,0.00),v40,z0,tPen\WObj:=wPaper;
    MoveL Offs(pOrigin,355.83,128.04,0.00),v40,z0,tPen\WObj:=wPaper;
    MoveL Offs(pOrigin,355.40,127.40,0.00),v40,z0,tPen\WObj:=wPaper;
    MoveL Offs(pOrigin,355.61,127.82,0.00),v40,z0,tPen\WObj:=wPaper;
    MoveL Offs(pOrigin,355.40,127.40,0.00),v40,fine,tPen\WObj:=wPaper;
    MoveL Offs(pOrigin,355.40,127.40,6.00),v60,z5,tPen\WObj:=wPaper;
    MoveL Offs(pOrigin,354.12,125.28,6.00),vTravel,z5,tPen\WObj:=wPaper;
    MoveL Offs(pOrigin,354.12,125.28,0.00),v60,z0,tPen\WObj:=wPaper;
    MoveL Offs(pOrigin,354.34,125.70,0.00),v40,z0,tPen\WObj:=wPaper;
    MoveL Offs(pOrigin,354.12,125.28,0.00),v40,fine,tPen\WObj:=wPaper;
    MoveL Offs(pOrigin,354.12,125.28,6.00),v60,z5,tPen\WObj:=wPaper;
    MoveL Offs(pOrigin,352.42,123.15,6.00),vTravel,z5,tPen\WObj:=wPaper;
    MoveL Offs(pOrigin,352.42,123.15,0.00),v60,z0,tPen\WObj:=wPaper;
    MoveL Offs(pOrigin,352.85,123.36,0.00),v40,z0,tPen\WObj:=wPaper;
    MoveL Offs(pOrigin,352.42,123.15,0.00),v40,z0,tPen\WObj:=wPaper;
    MoveL Offs(pOrigin,351.79,122.72,0.00),v40,z0,tPen\WObj:=wPaper;
    MoveL Offs(pOrigin,351.58,124.85,0.00),v40,z0,tPen\WObj:=wPaper;
    MoveL Offs(pOrigin,352.64,128.68,0.00),v40,fine,tPen\WObj:=wPaper;
    MoveL Offs(pOrigin,352.64,128.68,6.00),v60,z5,tPen\WObj:=wPaper;
    MoveL Offs(pOrigin,356.89,119.32,6.00),vTravel,z5,tPen\WObj:=wPaper;
    MoveL Offs(pOrigin,356.89,119.32,0.00),v60,z0,tPen\WObj:=wPaper;
    MoveL Offs(pOrigin,357.74,120.18,0.00),v40,z0,tPen\WObj:=wPaper;
    MoveL Offs(pOrigin,356.89,119.32,0.00),v40,fine,tPen\WObj:=wPaper;
    MoveL Offs(pOrigin,356.89,119.32,6.00),v60,z5,tPen\WObj:=wPaper;
    MoveL Offs(pOrigin,356.04,118.26,6.00),vTravel,z5,tPen\WObj:=wPaper;
    MoveL Offs(pOrigin,356.04,118.26,0.00),v60,z0,tPen\WObj:=wPaper;
    MoveL Offs(pOrigin,356.46,118.69,0.00),v40,z0,tPen\WObj:=wPaper;
    MoveL Offs(pOrigin,356.04,118.26,0.00),v40,fine,tPen\WObj:=wPaper;
    MoveL Offs(pOrigin,356.04,118.26,6.00),v60,z5,tPen\WObj:=wPaper;
    MoveL Offs(pOrigin,352.00,112.53,6.00),vTravel,z5,tPen\WObj:=wPaper;
    MoveL Offs(pOrigin,352.00,112.53,0.00),v60,z0,tPen\WObj:=wPaper;
    MoveL Offs(pOrigin,352.42,113.16,0.00),v40,z0,tPen\WObj:=wPaper;
    MoveL Offs(pOrigin,352.00,112.53,0.00),v40,fine,tPen\WObj:=wPaper;
    MoveL Offs(pOrigin,352.00,112.53,6.00),v60,z5,tPen\WObj:=wPaper;
    MoveL Offs(pOrigin,349.02,108.91,6.00),vTravel,z5,tPen\WObj:=wPaper;
    MoveL Offs(pOrigin,349.02,108.91,0.00),v60,z0,tPen\WObj:=wPaper;
    MoveL Offs(pOrigin,350.51,109.97,0.00),v40,z0,tPen\WObj:=wPaper;
    MoveL Offs(pOrigin,351.93,112.74,0.00),v40,z0,tPen\WObj:=wPaper;
    MoveL Offs(pOrigin,356.67,119.32,0.00),v40,z0,tPen\WObj:=wPaper;
    MoveL Offs(pOrigin,362.20,124.64,0.00),v40,z0,tPen\WObj:=wPaper;
    MoveL Offs(pOrigin,367.09,127.82,0.00),v40,fine,tPen\WObj:=wPaper;
    MoveL Offs(pOrigin,367.09,127.82,6.00),v60,z5,tPen\WObj:=wPaper;
    MoveL Offs(pOrigin,368.36,118.26,6.00),vTravel,z5,tPen\WObj:=wPaper;
    MoveL Offs(pOrigin,368.36,118.26,0.00),v60,z0,tPen\WObj:=wPaper;
    MoveL Offs(pOrigin,364.54,117.06,0.00),v40,z0,tPen\WObj:=wPaper;
    MoveL Offs(pOrigin,359.23,114.51,0.00),v40,z0,tPen\WObj:=wPaper;
    MoveL Offs(pOrigin,353.70,110.82,0.00),v40,z0,tPen\WObj:=wPaper;
    MoveL Offs(pOrigin,350.94,108.06,0.00),v40,z0,tPen\WObj:=wPaper;
    MoveL Offs(pOrigin,348.81,107.43,0.00),v40,fine,tPen\WObj:=wPaper;
    MoveL Offs(pOrigin,348.81,107.43,6.00),v60,z5,tPen\WObj:=wPaper;
    MoveL Offs(pOrigin,348.17,105.72,6.00),vTravel,z5,tPen\WObj:=wPaper;
    MoveL Offs(pOrigin,348.17,105.72,0.00),v60,z0,tPen\WObj:=wPaper;
    MoveL Offs(pOrigin,346.40,104.45,0.00),v40,z0,tPen\WObj:=wPaper;
    MoveL Offs(pOrigin,341.45,91.06,0.00),v40,z0,tPen\WObj:=wPaper;
    MoveL Offs(pOrigin,335.21,77.25,0.00),v40,fine,tPen\WObj:=wPaper;
    MoveL Offs(pOrigin,335.21,77.25,6.00),v60,z5,tPen\WObj:=wPaper;
    MoveL Offs(pOrigin,337.98,74.70,6.00),vTravel,z5,tPen\WObj:=wPaper;
    MoveL Offs(pOrigin,337.98,74.70,0.00),v60,z0,tPen\WObj:=wPaper;
    MoveL Offs(pOrigin,326.50,72.79,0.00),v40,z0,tPen\WObj:=wPaper;
    MoveL Offs(pOrigin,319.27,71.09,0.00),v40,z0,tPen\WObj:=wPaper;
    MoveL Offs(pOrigin,313.96,69.03,0.00),v40,z0,tPen\WObj:=wPaper;
    MoveL Offs(pOrigin,313.11,67.69,0.00),v40,z0,tPen\WObj:=wPaper;
  ENDPROC

  PROC DrawPart20()
    MoveL Offs(pOrigin,313.11,67.69,0.00),v40,z0,tPen\WObj:=wPaper;
    MoveL Offs(pOrigin,313.75,67.33,0.00),v40,z0,tPen\WObj:=wPaper;
    MoveL Offs(pOrigin,318.85,68.11,0.00),v40,z0,tPen\WObj:=wPaper;
    MoveL Offs(pOrigin,320.98,68.11,0.00),v40,z0,tPen\WObj:=wPaper;
    MoveL Offs(pOrigin,328.41,65.63,0.00),v40,z0,tPen\WObj:=wPaper;
    MoveL Offs(pOrigin,335.42,61.10,0.00),v40,z0,tPen\WObj:=wPaper;
    MoveL Offs(pOrigin,340.10,56.64,0.00),v40,z0,tPen\WObj:=wPaper;
    MoveL Offs(pOrigin,342.44,53.66,0.00),v40,z0,tPen\WObj:=wPaper;
    MoveL Offs(pOrigin,346.12,48.14,0.00),v40,z0,tPen\WObj:=wPaper;
    MoveL Offs(pOrigin,347.82,44.95,0.00),v40,z0,tPen\WObj:=wPaper;
    MoveL Offs(pOrigin,348.88,40.91,0.00),v40,z0,tPen\WObj:=wPaper;
    MoveL Offs(pOrigin,349.80,40.06,0.00),v40,z0,tPen\WObj:=wPaper;
    MoveL Offs(pOrigin,350.30,37.72,0.00),v40,z0,tPen\WObj:=wPaper;
    MoveL Offs(pOrigin,350.30,35.60,0.00),v40,z0,tPen\WObj:=wPaper;
    MoveL Offs(pOrigin,349.31,31.56,0.00),v40,z0,tPen\WObj:=wPaper;
    MoveL Offs(pOrigin,347.11,28.16,0.00),v40,z0,tPen\WObj:=wPaper;
    MoveL Offs(pOrigin,344.56,26.25,0.00),v40,z0,tPen\WObj:=wPaper;
    MoveL Offs(pOrigin,343.92,24.98,0.00),v40,fine,tPen\WObj:=wPaper;
    MoveL Offs(pOrigin,343.92,24.98,6.00),v60,z5,tPen\WObj:=wPaper;
    MoveL Offs(pOrigin,341.59,27.95,6.00),vTravel,z5,tPen\WObj:=wPaper;
    MoveL Offs(pOrigin,341.59,27.95,0.00),v60,z0,tPen\WObj:=wPaper;
    MoveL Offs(pOrigin,343.43,29.01,0.00),v40,z0,tPen\WObj:=wPaper;
    MoveL Offs(pOrigin,343.22,30.08,0.00),v40,z0,tPen\WObj:=wPaper;
    MoveL Offs(pOrigin,342.65,30.29,0.00),v40,z0,tPen\WObj:=wPaper;
    MoveL Offs(pOrigin,340.52,29.51,0.00),v40,z0,tPen\WObj:=wPaper;
    MoveL Offs(pOrigin,339.60,28.59,0.00),v40,z0,tPen\WObj:=wPaper;
    MoveL Offs(pOrigin,339.67,28.16,0.00),v40,z0,tPen\WObj:=wPaper;
    MoveL Offs(pOrigin,341.59,27.95,0.00),v40,fine,tPen\WObj:=wPaper;
    MoveL Offs(pOrigin,341.59,27.95,6.00),v60,z5,tPen\WObj:=wPaper;
    MoveL Offs(pOrigin,339.67,29.01,6.00),vTravel,z5,tPen\WObj:=wPaper;
    MoveL Offs(pOrigin,339.67,29.01,0.00),v60,z0,tPen\WObj:=wPaper;
    MoveL Offs(pOrigin,340.10,29.44,0.00),v40,z0,tPen\WObj:=wPaper;
    MoveL Offs(pOrigin,339.67,29.01,0.00),v40,z0,tPen\WObj:=wPaper;
    MoveL Offs(pOrigin,339.46,28.59,0.00),v40,z0,tPen\WObj:=wPaper;
    MoveL Offs(pOrigin,335.85,28.16,0.00),v40,z0,tPen\WObj:=wPaper;
    MoveL Offs(pOrigin,335.00,27.52,0.00),v40,fine,tPen\WObj:=wPaper;
    MoveL Offs(pOrigin,335.00,27.52,6.00),v60,z5,tPen\WObj:=wPaper;
    MoveL Offs(pOrigin,338.61,32.98,6.00),vTravel,z5,tPen\WObj:=wPaper;
    MoveL Offs(pOrigin,338.61,32.98,0.00),v60,z0,tPen\WObj:=wPaper;
    MoveL Offs(pOrigin,339.67,32.84,0.00),v40,z0,tPen\WObj:=wPaper;
    MoveL Offs(pOrigin,340.52,33.12,0.00),v40,z0,tPen\WObj:=wPaper;
    MoveL Offs(pOrigin,341.87,34.33,0.00),v40,z0,tPen\WObj:=wPaper;
    MoveL Offs(pOrigin,342.44,35.60,0.00),v40,z0,tPen\WObj:=wPaper;
    MoveL Offs(pOrigin,342.44,37.09,0.00),v40,z0,tPen\WObj:=wPaper;
    MoveL Offs(pOrigin,341.59,38.50,0.00),v40,z0,tPen\WObj:=wPaper;
    MoveL Offs(pOrigin,340.74,38.79,0.00),v40,z0,tPen\WObj:=wPaper;
    MoveL Offs(pOrigin,339.46,38.65,0.00),v40,z0,tPen\WObj:=wPaper;
    MoveL Offs(pOrigin,338.40,37.94,0.00),v40,z0,tPen\WObj:=wPaper;
    MoveL Offs(pOrigin,337.69,36.88,0.00),v40,z0,tPen\WObj:=wPaper;
    MoveL Offs(pOrigin,337.12,34.75,0.00),v40,z0,tPen\WObj:=wPaper;
    MoveL Offs(pOrigin,337.62,33.69,0.00),v40,z0,tPen\WObj:=wPaper;
    MoveL Offs(pOrigin,338.61,32.98,0.00),v40,fine,tPen\WObj:=wPaper;
    MoveL Offs(pOrigin,338.61,32.98,6.00),v60,z5,tPen\WObj:=wPaper;
    MoveL Offs(pOrigin,338.19,35.39,6.00),vTravel,z5,tPen\WObj:=wPaper;
    MoveL Offs(pOrigin,338.19,35.39,0.00),v60,z0,tPen\WObj:=wPaper;
    MoveL Offs(pOrigin,338.61,36.88,0.00),v40,z0,tPen\WObj:=wPaper;
    MoveL Offs(pOrigin,339.25,37.51,0.00),v40,fine,tPen\WObj:=wPaper;
    MoveL Offs(pOrigin,339.25,37.51,6.00),v60,z5,tPen\WObj:=wPaper;
    MoveL Offs(pOrigin,341.16,38.79,6.00),vTravel,z5,tPen\WObj:=wPaper;
    MoveL Offs(pOrigin,341.16,38.79,0.00),v60,z0,tPen\WObj:=wPaper;
    MoveL Offs(pOrigin,341.59,38.36,0.00),v40,z0,tPen\WObj:=wPaper;
    MoveL Offs(pOrigin,341.16,38.79,0.00),v40,fine,tPen\WObj:=wPaper;
    MoveL Offs(pOrigin,341.16,38.79,6.00),v60,z5,tPen\WObj:=wPaper;
    MoveL Offs(pOrigin,342.01,34.33,6.00),vTravel,z5,tPen\WObj:=wPaper;
    MoveL Offs(pOrigin,342.01,34.33,0.00),v60,z0,tPen\WObj:=wPaper;
    MoveL Offs(pOrigin,342.23,34.75,0.00),v40,z0,tPen\WObj:=wPaper;
    MoveL Offs(pOrigin,342.01,34.33,0.00),v40,fine,tPen\WObj:=wPaper;
    MoveL Offs(pOrigin,342.01,34.33,6.00),v60,z5,tPen\WObj:=wPaper;
    MoveL Offs(pOrigin,343.50,30.08,6.00),vTravel,z5,tPen\WObj:=wPaper;
    MoveL Offs(pOrigin,343.50,30.08,0.00),v60,z0,tPen\WObj:=wPaper;
    MoveL Offs(pOrigin,345.20,31.56,0.00),v40,z0,tPen\WObj:=wPaper;
    MoveL Offs(pOrigin,346.55,33.69,0.00),v40,z0,tPen\WObj:=wPaper;
    MoveL Offs(pOrigin,347.75,36.88,0.00),v40,z0,tPen\WObj:=wPaper;
    MoveL Offs(pOrigin,348.17,39.64,0.00),v40,z0,tPen\WObj:=wPaper;
    MoveL Offs(pOrigin,348.81,40.70,0.00),v40,z0,tPen\WObj:=wPaper;
    MoveL Offs(pOrigin,348.81,40.70,0.00),v40,z0,tPen\WObj:=wPaper;
    MoveL Offs(pOrigin,348.17,40.06,0.00),v40,fine,tPen\WObj:=wPaper;
    MoveL Offs(pOrigin,348.17,40.06,6.00),v60,z5,tPen\WObj:=wPaper;
    MoveL Offs(pOrigin,354.55,39.42,6.00),vTravel,z5,tPen\WObj:=wPaper;
    MoveL Offs(pOrigin,354.55,39.42,0.00),v60,z0,tPen\WObj:=wPaper;
    MoveL Offs(pOrigin,353.91,36.24,0.00),v40,z0,tPen\WObj:=wPaper;
    MoveL Offs(pOrigin,352.85,33.47,0.00),v40,z0,tPen\WObj:=wPaper;
    MoveL Offs(pOrigin,353.06,34.33,0.00),v40,z0,tPen\WObj:=wPaper;
    MoveL Offs(pOrigin,353.27,34.75,0.00),v40,z0,tPen\WObj:=wPaper;
    MoveL Offs(pOrigin,353.06,34.33,0.00),v40,fine,tPen\WObj:=wPaper;
    MoveL Offs(pOrigin,353.06,34.33,6.00),v60,z5,tPen\WObj:=wPaper;
    MoveL Offs(pOrigin,358.38,29.86,6.00),vTravel,z5,tPen\WObj:=wPaper;
    MoveL Offs(pOrigin,358.38,29.86,0.00),v60,z0,tPen\WObj:=wPaper;
    MoveL Offs(pOrigin,358.80,30.08,0.00),v40,z0,tPen\WObj:=wPaper;
    MoveL Offs(pOrigin,358.38,29.86,0.00),v40,fine,tPen\WObj:=wPaper;
    MoveL Offs(pOrigin,358.38,29.86,6.00),v60,z5,tPen\WObj:=wPaper;
    MoveL Offs(pOrigin,365.60,32.20,6.00),vTravel,z5,tPen\WObj:=wPaper;
    MoveL Offs(pOrigin,365.60,32.20,0.00),v60,z0,tPen\WObj:=wPaper;
    MoveL Offs(pOrigin,366.66,33.55,0.00),v40,z0,tPen\WObj:=wPaper;
    MoveL Offs(pOrigin,370.06,34.82,0.00),v40,z0,tPen\WObj:=wPaper;
    MoveL Offs(pOrigin,381.96,38.36,0.00),v40,z0,tPen\WObj:=wPaper;
    MoveL Offs(pOrigin,384.09,38.58,0.00),v40,fine,tPen\WObj:=wPaper;
    MoveL Offs(pOrigin,384.09,38.58,6.00),v60,z5,tPen\WObj:=wPaper;
    MoveL Offs(pOrigin,384.30,46.44,6.00),vTravel,z5,tPen\WObj:=wPaper;
    MoveL Offs(pOrigin,384.30,46.44,0.00),v60,z0,tPen\WObj:=wPaper;
    MoveL Offs(pOrigin,377.71,52.81,0.00),v40,z0,tPen\WObj:=wPaper;
    MoveL Offs(pOrigin,377.29,53.03,0.00),v40,z0,tPen\WObj:=wPaper;
    MoveL Offs(pOrigin,371.55,57.91,0.00),v40,fine,tPen\WObj:=wPaper;
    MoveL Offs(pOrigin,371.55,57.91,6.00),v60,z5,tPen\WObj:=wPaper;
    MoveL Offs(pOrigin,377.08,58.34,6.00),vTravel,z5,tPen\WObj:=wPaper;
    MoveL Offs(pOrigin,377.08,58.34,0.00),v60,z0,tPen\WObj:=wPaper;
    MoveL Offs(pOrigin,376.65,58.76,0.00),v40,z0,tPen\WObj:=wPaper;
    MoveL Offs(pOrigin,377.08,58.34,0.00),v40,z0,tPen\WObj:=wPaper;
    MoveL Offs(pOrigin,377.92,57.70,0.00),v40,z0,tPen\WObj:=wPaper;
    MoveL Offs(pOrigin,374.74,60.46,0.00),v40,z0,tPen\WObj:=wPaper;
    MoveL Offs(pOrigin,370.91,63.08,0.00),v40,z0,tPen\WObj:=wPaper;
    MoveL Offs(pOrigin,361.56,67.97,0.00),v40,z0,tPen\WObj:=wPaper;
    MoveL Offs(pOrigin,355.19,70.24,0.00),v40,z0,tPen\WObj:=wPaper;
    MoveL Offs(pOrigin,349.66,71.72,0.00),v40,z0,tPen\WObj:=wPaper;
    MoveL Offs(pOrigin,341.80,72.79,0.00),v40,fine,tPen\WObj:=wPaper;
    MoveL Offs(pOrigin,341.80,72.79,6.00),v60,z5,tPen\WObj:=wPaper;
    MoveL Offs(pOrigin,337.98,74.70,6.00),vTravel,z5,tPen\WObj:=wPaper;
    MoveL Offs(pOrigin,337.98,74.70,0.00),v60,z0,tPen\WObj:=wPaper;
    MoveL Offs(pOrigin,346.90,75.76,0.00),v40,z0,tPen\WObj:=wPaper;
    MoveL Offs(pOrigin,347.75,76.19,0.00),v40,z0,tPen\WObj:=wPaper;
  ENDPROC

  PROC DrawPart21()
    MoveL Offs(pOrigin,347.75,76.19,0.00),v40,z0,tPen\WObj:=wPaper;
    MoveL Offs(pOrigin,349.24,87.45,0.00),v40,z0,tPen\WObj:=wPaper;
    MoveL Offs(pOrigin,349.45,91.70,0.00),v40,z0,tPen\WObj:=wPaper;
    MoveL Offs(pOrigin,349.88,92.34,0.00),v40,z0,tPen\WObj:=wPaper;
    MoveL Offs(pOrigin,349.88,92.34,0.00),v40,z0,tPen\WObj:=wPaper;
    MoveL Offs(pOrigin,348.39,96.59,0.00),v40,z0,tPen\WObj:=wPaper;
    MoveL Offs(pOrigin,348.17,98.50,0.00),v40,z0,tPen\WObj:=wPaper;
    MoveL Offs(pOrigin,347.75,99.14,0.00),v40,z0,tPen\WObj:=wPaper;
    MoveL Offs(pOrigin,347.75,99.14,0.00),v40,z0,tPen\WObj:=wPaper;
    MoveL Offs(pOrigin,348.17,101.47,0.00),v40,fine,tPen\WObj:=wPaper;
    MoveL Offs(pOrigin,348.17,101.47,6.00),v60,z5,tPen\WObj:=wPaper;
    MoveL Offs(pOrigin,347.75,99.14,6.00),vTravel,z5,tPen\WObj:=wPaper;
    MoveL Offs(pOrigin,347.75,99.14,0.00),v60,z0,tPen\WObj:=wPaper;
    MoveL Offs(pOrigin,346.62,98.50,0.00),v40,z0,tPen\WObj:=wPaper;
    MoveL Offs(pOrigin,344.00,90.00,0.00),v40,z0,tPen\WObj:=wPaper;
    MoveL Offs(pOrigin,341.02,82.14,0.00),v40,z0,tPen\WObj:=wPaper;
    MoveL Offs(pOrigin,338.12,76.19,0.00),v40,z0,tPen\WObj:=wPaper;
    MoveL Offs(pOrigin,337.98,74.70,0.00),v40,fine,tPen\WObj:=wPaper;
    MoveL Offs(pOrigin,337.98,74.70,6.00),v60,z5,tPen\WObj:=wPaper;
    MoveL Offs(pOrigin,339.46,78.53,6.00),vTravel,z5,tPen\WObj:=wPaper;
    MoveL Offs(pOrigin,339.46,78.53,0.00),v60,z0,tPen\WObj:=wPaper;
    MoveL Offs(pOrigin,339.67,78.95,0.00),v40,z0,tPen\WObj:=wPaper;
    MoveL Offs(pOrigin,339.46,78.53,0.00),v40,fine,tPen\WObj:=wPaper;
    MoveL Offs(pOrigin,339.46,78.53,6.00),v60,z5,tPen\WObj:=wPaper;
    MoveL Offs(pOrigin,337.12,81.71,6.00),vTravel,z5,tPen\WObj:=wPaper;
    MoveL Offs(pOrigin,337.12,81.71,0.00),v60,z0,tPen\WObj:=wPaper;
    MoveL Offs(pOrigin,337.34,82.14,0.00),v40,z0,tPen\WObj:=wPaper;
    MoveL Offs(pOrigin,337.12,81.71,0.00),v40,fine,tPen\WObj:=wPaper;
    MoveL Offs(pOrigin,337.12,81.71,6.00),v60,z5,tPen\WObj:=wPaper;
    MoveL Offs(pOrigin,337.76,83.20,6.00),vTravel,z5,tPen\WObj:=wPaper;
    MoveL Offs(pOrigin,337.76,83.20,0.00),v60,z0,tPen\WObj:=wPaper;
    MoveL Offs(pOrigin,337.98,83.62,0.00),v40,z0,tPen\WObj:=wPaper;
    MoveL Offs(pOrigin,337.76,83.20,0.00),v40,fine,tPen\WObj:=wPaper;
    MoveL Offs(pOrigin,337.76,83.20,6.00),v60,z5,tPen\WObj:=wPaper;
    MoveL Offs(pOrigin,347.75,76.19,6.00),vTravel,z5,tPen\WObj:=wPaper;
    MoveL Offs(pOrigin,347.75,76.19,0.00),v60,z0,tPen\WObj:=wPaper;
    MoveL Offs(pOrigin,348.60,75.97,0.00),v40,z0,tPen\WObj:=wPaper;
    MoveL Offs(pOrigin,352.21,76.40,0.00),v40,z0,tPen\WObj:=wPaper;
    MoveL Offs(pOrigin,353.27,76.82,0.00),v40,fine,tPen\WObj:=wPaper;
    MoveL Offs(pOrigin,353.27,76.82,6.00),v60,z5,tPen\WObj:=wPaper;
    MoveL Offs(pOrigin,355.61,78.31,6.00),vTravel,z5,tPen\WObj:=wPaper;
    MoveL Offs(pOrigin,355.61,78.31,0.00),v60,z0,tPen\WObj:=wPaper;
    MoveL Offs(pOrigin,357.31,81.29,0.00),v40,z0,tPen\WObj:=wPaper;
    MoveL Offs(pOrigin,359.65,84.26,0.00),v40,z0,tPen\WObj:=wPaper;
    MoveL Offs(pOrigin,363.48,88.09,0.00),v40,z0,tPen\WObj:=wPaper;
    MoveL Offs(pOrigin,367.09,90.64,0.00),v40,fine,tPen\WObj:=wPaper;
    MoveL Offs(pOrigin,367.09,90.64,6.00),v60,z5,tPen\WObj:=wPaper;
    MoveL Offs(pOrigin,363.26,87.66,6.00),vTravel,z5,tPen\WObj:=wPaper;
    MoveL Offs(pOrigin,363.26,87.66,0.00),v60,z0,tPen\WObj:=wPaper;
    MoveL Offs(pOrigin,363.69,88.09,0.00),v40,z0,tPen\WObj:=wPaper;
    MoveL Offs(pOrigin,363.26,87.66,0.00),v40,fine,tPen\WObj:=wPaper;
    MoveL Offs(pOrigin,363.26,87.66,6.00),v60,z5,tPen\WObj:=wPaper;
    MoveL Offs(pOrigin,360.08,88.94,6.00),vTravel,z5,tPen\WObj:=wPaper;
    MoveL Offs(pOrigin,360.08,88.94,0.00),v60,z0,tPen\WObj:=wPaper;
    MoveL Offs(pOrigin,361.14,90.00,0.00),v40,z0,tPen\WObj:=wPaper;
    MoveL Offs(pOrigin,360.08,88.94,0.00),v40,fine,tPen\WObj:=wPaper;
    MoveL Offs(pOrigin,360.08,88.94,6.00),v60,z5,tPen\WObj:=wPaper;
    MoveL Offs(pOrigin,357.52,85.54,6.00),vTravel,z5,tPen\WObj:=wPaper;
    MoveL Offs(pOrigin,357.52,85.54,0.00),v60,z0,tPen\WObj:=wPaper;
    MoveL Offs(pOrigin,360.08,89.15,0.00),v40,z0,tPen\WObj:=wPaper;
    MoveL Offs(pOrigin,364.75,93.40,0.00),v40,z0,tPen\WObj:=wPaper;
    MoveL Offs(pOrigin,369.42,96.02,0.00),v40,z0,tPen\WObj:=wPaper;
    MoveL Offs(pOrigin,373.25,97.01,0.00),v40,fine,tPen\WObj:=wPaper;
    MoveL Offs(pOrigin,373.25,97.01,6.00),v60,z5,tPen\WObj:=wPaper;
    MoveL Offs(pOrigin,378.99,87.45,6.00),vTravel,z5,tPen\WObj:=wPaper;
    MoveL Offs(pOrigin,378.99,87.45,0.00),v60,z0,tPen\WObj:=wPaper;
    MoveL Offs(pOrigin,382.17,88.72,0.00),v40,z0,tPen\WObj:=wPaper;
    MoveL Offs(pOrigin,387.70,89.79,0.00),v40,z0,tPen\WObj:=wPaper;
    MoveL Offs(pOrigin,393.44,89.79,0.00),v40,z0,tPen\WObj:=wPaper;
    MoveL Offs(pOrigin,396.41,89.15,0.00),v40,fine,tPen\WObj:=wPaper;
    MoveL Offs(pOrigin,396.41,89.15,6.00),v60,z5,tPen\WObj:=wPaper;
    MoveL Offs(pOrigin,403.85,94.25,6.00),vTravel,z5,tPen\WObj:=wPaper;
    MoveL Offs(pOrigin,403.85,94.25,0.00),v60,z0,tPen\WObj:=wPaper;
    MoveL Offs(pOrigin,400.45,97.22,0.00),v40,z0,tPen\WObj:=wPaper;
    MoveL Offs(pOrigin,394.29,100.70,0.00),v40,z0,tPen\WObj:=wPaper;
    MoveL Offs(pOrigin,386.64,103.39,0.00),v40,z0,tPen\WObj:=wPaper;
    MoveL Offs(pOrigin,383.02,104.24,0.00),v40,z0,tPen\WObj:=wPaper;
    MoveL Offs(pOrigin,377.92,104.88,0.00),v40,z0,tPen\WObj:=wPaper;
    MoveL Offs(pOrigin,371.12,104.66,0.00),v40,z0,tPen\WObj:=wPaper;
    MoveL Offs(pOrigin,365.60,103.03,0.00),v40,z0,tPen\WObj:=wPaper;
    MoveL Offs(pOrigin,361.56,100.20,0.00),v40,z0,tPen\WObj:=wPaper;
    MoveL Offs(pOrigin,359.65,97.01,0.00),v40,fine,tPen\WObj:=wPaper;
    MoveL Offs(pOrigin,359.65,97.01,6.00),v60,z5,tPen\WObj:=wPaper;
    MoveL Offs(pOrigin,360.92,99.14,6.00),vTravel,z5,tPen\WObj:=wPaper;
    MoveL Offs(pOrigin,360.92,99.14,0.00),v60,z0,tPen\WObj:=wPaper;
    MoveL Offs(pOrigin,361.35,99.56,0.00),v40,z0,tPen\WObj:=wPaper;
    MoveL Offs(pOrigin,360.92,99.14,0.00),v40,fine,tPen\WObj:=wPaper;
    MoveL Offs(pOrigin,360.92,99.14,6.00),v60,z5,tPen\WObj:=wPaper;
    MoveL Offs(pOrigin,361.77,100.20,6.00),vTravel,z5,tPen\WObj:=wPaper;
    MoveL Offs(pOrigin,361.77,100.20,0.00),v60,z0,tPen\WObj:=wPaper;
    MoveL Offs(pOrigin,362.41,100.84,0.00),v40,z0,tPen\WObj:=wPaper;
    MoveL Offs(pOrigin,361.77,100.20,0.00),v40,fine,tPen\WObj:=wPaper;
    MoveL Offs(pOrigin,361.77,100.20,6.00),v60,z5,tPen\WObj:=wPaper;
    MoveL Offs(pOrigin,356.25,99.78,6.00),vTravel,z5,tPen\WObj:=wPaper;
    MoveL Offs(pOrigin,356.25,99.78,0.00),v60,z0,tPen\WObj:=wPaper;
    MoveL Offs(pOrigin,354.05,95.74,0.00),v40,z0,tPen\WObj:=wPaper;
    MoveL Offs(pOrigin,353.06,91.28,0.00),v40,z0,tPen\WObj:=wPaper;
    MoveL Offs(pOrigin,352.21,90.00,0.00),v40,z0,tPen\WObj:=wPaper;
    MoveL Offs(pOrigin,352.64,81.71,0.00),v40,z0,tPen\WObj:=wPaper;
    MoveL Offs(pOrigin,353.27,77.25,0.00),v40,z0,tPen\WObj:=wPaper;
    MoveL Offs(pOrigin,353.70,76.68,0.00),v40,z0,tPen\WObj:=wPaper;
    MoveL Offs(pOrigin,361.56,77.32,0.00),v40,z0,tPen\WObj:=wPaper;
    MoveL Offs(pOrigin,362.20,78.31,0.00),v40,z0,tPen\WObj:=wPaper;
    MoveL Offs(pOrigin,367.30,81.36,0.00),v40,z0,tPen\WObj:=wPaper;
    MoveL Offs(pOrigin,370.91,83.06,0.00),v40,z0,tPen\WObj:=wPaper;
    MoveL Offs(pOrigin,375.16,84.47,0.00),v40,z0,tPen\WObj:=wPaper;
    MoveL Offs(pOrigin,378.77,85.11,0.00),v40,z0,tPen\WObj:=wPaper;
    MoveL Offs(pOrigin,381.54,85.11,0.00),v40,z0,tPen\WObj:=wPaper;
    MoveL Offs(pOrigin,383.45,86.18,0.00),v40,z0,tPen\WObj:=wPaper;
    MoveL Offs(pOrigin,388.34,86.18,0.00),v40,z0,tPen\WObj:=wPaper;
    MoveL Offs(pOrigin,394.50,84.90,0.00),v40,z0,tPen\WObj:=wPaper;
    MoveL Offs(pOrigin,400.45,82.42,0.00),v40,z0,tPen\WObj:=wPaper;
    MoveL Offs(pOrigin,406.19,78.31,0.00),v40,z0,tPen\WObj:=wPaper;
    MoveL Offs(pOrigin,410.01,74.49,0.00),v40,z0,tPen\WObj:=wPaper;
    MoveL Offs(pOrigin,410.86,73.21,0.00),v40,fine,tPen\WObj:=wPaper;
    MoveL Offs(pOrigin,410.86,73.21,6.00),v60,z5,tPen\WObj:=wPaper;
    MoveL Offs(pOrigin,410.01,74.28,6.00),vTravel,z5,tPen\WObj:=wPaper;
    MoveL Offs(pOrigin,410.01,74.28,0.00),v60,z0,tPen\WObj:=wPaper;
    MoveL Offs(pOrigin,409.38,74.91,0.00),v40,z0,tPen\WObj:=wPaper;
    MoveL Offs(pOrigin,410.01,74.28,0.00),v40,fine,tPen\WObj:=wPaper;
  ENDPROC

  PROC DrawPart22()
    MoveL Offs(pOrigin,410.01,74.28,6.00),v60,z5,tPen\WObj:=wPaper;
    MoveL Offs(pOrigin,406.40,73.85,6.00),vTravel,z5,tPen\WObj:=wPaper;
    MoveL Offs(pOrigin,406.40,73.85,0.00),v60,z0,tPen\WObj:=wPaper;
    MoveL Offs(pOrigin,411.22,69.60,0.00),v40,z0,tPen\WObj:=wPaper;
    MoveL Offs(pOrigin,413.62,66.48,0.00),v40,z0,tPen\WObj:=wPaper;
    MoveL Offs(pOrigin,414.69,65.99,0.00),v40,fine,tPen\WObj:=wPaper;
    MoveL Offs(pOrigin,414.69,65.99,6.00),v60,z5,tPen\WObj:=wPaper;
    MoveL Offs(pOrigin,412.35,68.11,6.00),vTravel,z5,tPen\WObj:=wPaper;
    MoveL Offs(pOrigin,412.35,68.11,0.00),v60,z0,tPen\WObj:=wPaper;
    MoveL Offs(pOrigin,412.14,68.54,0.00),v40,z0,tPen\WObj:=wPaper;
    MoveL Offs(pOrigin,412.35,68.11,0.00),v40,fine,tPen\WObj:=wPaper;
    MoveL Offs(pOrigin,412.35,68.11,6.00),v60,z5,tPen\WObj:=wPaper;
    MoveL Offs(pOrigin,411.08,69.60,6.00),vTravel,z5,tPen\WObj:=wPaper;
    MoveL Offs(pOrigin,411.08,69.60,0.00),v60,z0,tPen\WObj:=wPaper;
    MoveL Offs(pOrigin,410.86,70.03,0.00),v40,z0,tPen\WObj:=wPaper;
    MoveL Offs(pOrigin,411.08,69.60,0.00),v40,fine,tPen\WObj:=wPaper;
    MoveL Offs(pOrigin,411.08,69.60,6.00),v60,z5,tPen\WObj:=wPaper;
    MoveL Offs(pOrigin,407.25,67.26,6.00),vTravel,z5,tPen\WObj:=wPaper;
    MoveL Offs(pOrigin,407.25,67.26,0.00),v60,z0,tPen\WObj:=wPaper;
    MoveL Offs(pOrigin,404.70,70.88,0.00),v40,fine,tPen\WObj:=wPaper;
    MoveL Offs(pOrigin,404.70,70.88,6.00),v60,z5,tPen\WObj:=wPaper;
    MoveL Offs(pOrigin,405.55,69.60,6.00),vTravel,z5,tPen\WObj:=wPaper;
    MoveL Offs(pOrigin,405.55,69.60,0.00),v60,z0,tPen\WObj:=wPaper;
    MoveL Offs(pOrigin,405.34,70.03,0.00),v40,z0,tPen\WObj:=wPaper;
    MoveL Offs(pOrigin,405.55,69.60,0.00),v40,z0,tPen\WObj:=wPaper;
    MoveL Offs(pOrigin,406.19,68.75,0.00),v40,z0,tPen\WObj:=wPaper;
    MoveL Offs(pOrigin,405.98,69.18,0.00),v40,z0,tPen\WObj:=wPaper;
    MoveL Offs(pOrigin,406.19,68.75,0.00),v40,fine,tPen\WObj:=wPaper;
    MoveL Offs(pOrigin,406.19,68.75,6.00),v60,z5,tPen\WObj:=wPaper;
    MoveL Offs(pOrigin,405.98,66.20,6.00),vTravel,z5,tPen\WObj:=wPaper;
    MoveL Offs(pOrigin,405.98,66.20,0.00),v60,z0,tPen\WObj:=wPaper;
    MoveL Offs(pOrigin,405.76,66.62,0.00),v40,z0,tPen\WObj:=wPaper;
    MoveL Offs(pOrigin,405.98,66.20,0.00),v40,z0,tPen\WObj:=wPaper;
    MoveL Offs(pOrigin,406.40,65.35,0.00),v40,z0,tPen\WObj:=wPaper;
    MoveL Offs(pOrigin,406.19,65.78,0.00),v40,z0,tPen\WObj:=wPaper;
    MoveL Offs(pOrigin,406.40,65.35,0.00),v40,fine,tPen\WObj:=wPaper;
    MoveL Offs(pOrigin,406.40,65.35,6.00),v60,z5,tPen\WObj:=wPaper;
    MoveL Offs(pOrigin,403.00,71.30,6.00),vTravel,z5,tPen\WObj:=wPaper;
    MoveL Offs(pOrigin,403.00,71.30,0.00),v60,z0,tPen\WObj:=wPaper;
    MoveL Offs(pOrigin,406.68,65.14,0.00),v40,z0,tPen\WObj:=wPaper;
    MoveL Offs(pOrigin,408.17,61.53,0.00),v40,z0,tPen\WObj:=wPaper;
    MoveL Offs(pOrigin,409.59,56.64,0.00),v40,z0,tPen\WObj:=wPaper;
    MoveL Offs(pOrigin,409.80,48.56,0.00),v40,z0,tPen\WObj:=wPaper;
    MoveL Offs(pOrigin,407.89,41.76,0.00),v40,z0,tPen\WObj:=wPaper;
    MoveL Offs(pOrigin,408.10,41.34,0.00),v40,fine,tPen\WObj:=wPaper;
    MoveL Offs(pOrigin,408.10,41.34,6.00),v60,z5,tPen\WObj:=wPaper;
    MoveL Offs(pOrigin,402.36,43.67,6.00),vTravel,z5,tPen\WObj:=wPaper;
    MoveL Offs(pOrigin,402.36,43.67,0.00),v60,z0,tPen\WObj:=wPaper;
    MoveL Offs(pOrigin,401.30,49.84,0.00),v40,z0,tPen\WObj:=wPaper;
    MoveL Offs(pOrigin,399.46,54.51,0.00),v40,z0,tPen\WObj:=wPaper;
    MoveL Offs(pOrigin,395.99,60.25,0.00),v40,z0,tPen\WObj:=wPaper;
    MoveL Offs(pOrigin,391.31,65.78,0.00),v40,z0,tPen\WObj:=wPaper;
    MoveL Offs(pOrigin,390.89,65.99,0.00),v40,z0,tPen\WObj:=wPaper;
    MoveL Offs(pOrigin,387.91,68.75,0.00),v40,z0,tPen\WObj:=wPaper;
    MoveL Offs(pOrigin,383.88,71.58,0.00),v40,z0,tPen\WObj:=wPaper;
    MoveL Offs(pOrigin,377.92,74.56,0.00),v40,z0,tPen\WObj:=wPaper;
    MoveL Offs(pOrigin,372.83,75.97,0.00),v40,z0,tPen\WObj:=wPaper;
    MoveL Offs(pOrigin,366.88,76.82,0.00),v40,z0,tPen\WObj:=wPaper;
    MoveL Offs(pOrigin,362.41,76.82,0.00),v40,z0,tPen\WObj:=wPaper;
    MoveL Offs(pOrigin,361.77,77.25,0.00),v40,fine,tPen\WObj:=wPaper;
    MoveL Offs(pOrigin,361.77,77.25,6.00),v60,z5,tPen\WObj:=wPaper;
    MoveL Offs(pOrigin,367.09,79.59,6.00),vTravel,z5,tPen\WObj:=wPaper;
    MoveL Offs(pOrigin,367.09,79.59,0.00),v60,z0,tPen\WObj:=wPaper;
    MoveL Offs(pOrigin,369.42,80.22,0.00),v40,z0,tPen\WObj:=wPaper;
    MoveL Offs(pOrigin,376.23,80.44,0.00),v40,z0,tPen\WObj:=wPaper;
    MoveL Offs(pOrigin,381.33,79.80,0.00),v40,z0,tPen\WObj:=wPaper;
    MoveL Offs(pOrigin,385.79,78.53,0.00),v40,fine,tPen\WObj:=wPaper;
    MoveL Offs(pOrigin,385.79,78.53,6.00),v60,z5,tPen\WObj:=wPaper;
    MoveL Offs(pOrigin,381.96,85.11,6.00),vTravel,z5,tPen\WObj:=wPaper;
    MoveL Offs(pOrigin,381.96,85.11,0.00),v60,z0,tPen\WObj:=wPaper;
    MoveL Offs(pOrigin,383.24,84.26,0.00),v40,z0,tPen\WObj:=wPaper;
    MoveL Offs(pOrigin,389.19,82.99,0.00),v40,z0,tPen\WObj:=wPaper;
    MoveL Offs(pOrigin,394.50,80.93,0.00),v40,z0,tPen\WObj:=wPaper;
    MoveL Offs(pOrigin,400.24,77.96,0.00),v40,z0,tPen\WObj:=wPaper;
    MoveL Offs(pOrigin,405.98,74.06,0.00),v40,fine,tPen\WObj:=wPaper;
    MoveL Offs(pOrigin,405.98,74.06,6.00),v60,z5,tPen\WObj:=wPaper;
    MoveL Offs(pOrigin,412.35,77.89,6.00),vTravel,z5,tPen\WObj:=wPaper;
    MoveL Offs(pOrigin,412.35,77.89,0.00),v60,z0,tPen\WObj:=wPaper;
    MoveL Offs(pOrigin,412.14,78.31,0.00),v40,z0,tPen\WObj:=wPaper;
    MoveL Offs(pOrigin,412.35,77.89,0.00),v40,fine,tPen\WObj:=wPaper;
    MoveL Offs(pOrigin,412.35,77.89,6.00),v60,z5,tPen\WObj:=wPaper;
    MoveL Offs(pOrigin,393.86,62.80,6.00),vTravel,z5,tPen\WObj:=wPaper;
    MoveL Offs(pOrigin,393.86,62.80,0.00),v60,z0,tPen\WObj:=wPaper;
    MoveL Offs(pOrigin,393.65,63.22,0.00),v40,z0,tPen\WObj:=wPaper;
    MoveL Offs(pOrigin,393.86,62.80,0.00),v40,fine,tPen\WObj:=wPaper;
    MoveL Offs(pOrigin,393.86,62.80,6.00),v60,z5,tPen\WObj:=wPaper;
    MoveL Offs(pOrigin,394.71,61.74,6.00),vTravel,z5,tPen\WObj:=wPaper;
    MoveL Offs(pOrigin,394.71,61.74,0.00),v60,z0,tPen\WObj:=wPaper;
    MoveL Offs(pOrigin,394.50,62.16,0.00),v40,z0,tPen\WObj:=wPaper;
    MoveL Offs(pOrigin,394.71,61.74,0.00),v40,fine,tPen\WObj:=wPaper;
    MoveL Offs(pOrigin,394.71,61.74,6.00),v60,z5,tPen\WObj:=wPaper;
    MoveL Offs(pOrigin,392.16,64.71,6.00),vTravel,z5,tPen\WObj:=wPaper;
    MoveL Offs(pOrigin,392.16,64.71,0.00),v60,z0,tPen\WObj:=wPaper;
    MoveL Offs(pOrigin,391.95,65.14,0.00),v40,z0,tPen\WObj:=wPaper;
    MoveL Offs(pOrigin,392.16,64.71,0.00),v40,fine,tPen\WObj:=wPaper;
    MoveL Offs(pOrigin,392.16,64.71,6.00),v60,z5,tPen\WObj:=wPaper;
    MoveL Offs(pOrigin,389.61,67.05,6.00),vTravel,z5,tPen\WObj:=wPaper;
    MoveL Offs(pOrigin,389.61,67.05,0.00),v60,z0,tPen\WObj:=wPaper;
    MoveL Offs(pOrigin,388.98,67.69,0.00),v40,z0,tPen\WObj:=wPaper;
    MoveL Offs(pOrigin,389.61,67.05,0.00),v40,fine,tPen\WObj:=wPaper;
    MoveL Offs(pOrigin,389.61,67.05,6.00),v60,z5,tPen\WObj:=wPaper;
    MoveL Offs(pOrigin,397.90,57.06,6.00),vTravel,z5,tPen\WObj:=wPaper;
    MoveL Offs(pOrigin,397.90,57.06,0.00),v60,z0,tPen\WObj:=wPaper;
    MoveL Offs(pOrigin,397.69,57.49,0.00),v40,z0,tPen\WObj:=wPaper;
    MoveL Offs(pOrigin,397.90,57.06,0.00),v40,fine,tPen\WObj:=wPaper;
    MoveL Offs(pOrigin,397.90,57.06,6.00),v60,z5,tPen\WObj:=wPaper;
    MoveL Offs(pOrigin,398.75,55.58,6.00),vTravel,z5,tPen\WObj:=wPaper;
    MoveL Offs(pOrigin,398.75,55.58,0.00),v60,z0,tPen\WObj:=wPaper;
    MoveL Offs(pOrigin,398.54,56.00,0.00),v40,z0,tPen\WObj:=wPaper;
    MoveL Offs(pOrigin,398.75,55.58,0.00),v40,fine,tPen\WObj:=wPaper;
    MoveL Offs(pOrigin,398.75,55.58,6.00),v60,z5,tPen\WObj:=wPaper;
    MoveL Offs(pOrigin,399.81,53.45,6.00),vTravel,z5,tPen\WObj:=wPaper;
    MoveL Offs(pOrigin,399.81,53.45,0.00),v60,z0,tPen\WObj:=wPaper;
    MoveL Offs(pOrigin,399.60,53.88,0.00),v40,z0,tPen\WObj:=wPaper;
    MoveL Offs(pOrigin,399.81,53.45,0.00),v40,fine,tPen\WObj:=wPaper;
    MoveL Offs(pOrigin,399.81,53.45,6.00),v60,z5,tPen\WObj:=wPaper;
    MoveL Offs(pOrigin,383.02,52.81,6.00),vTravel,z5,tPen\WObj:=wPaper;
    MoveL Offs(pOrigin,383.02,52.81,0.00),v60,z0,tPen\WObj:=wPaper;
    MoveL Offs(pOrigin,378.35,57.49,0.00),v40,fine,tPen\WObj:=wPaper;
    MoveL Offs(pOrigin,378.35,57.49,6.00),v60,z5,tPen\WObj:=wPaper;
  ENDPROC

  PROC DrawPart23()
    MoveL Offs(pOrigin,378.56,51.75,6.00),vTravel,z5,tPen\WObj:=wPaper;
    MoveL Offs(pOrigin,378.56,51.75,0.00),v60,z0,tPen\WObj:=wPaper;
    MoveL Offs(pOrigin,378.35,52.17,0.00),v40,z0,tPen\WObj:=wPaper;
    MoveL Offs(pOrigin,378.56,51.75,0.00),v40,z0,tPen\WObj:=wPaper;
    MoveL Offs(pOrigin,379.20,51.11,0.00),v40,z0,tPen\WObj:=wPaper;
    MoveL Offs(pOrigin,378.99,51.54,0.00),v40,z0,tPen\WObj:=wPaper;
    MoveL Offs(pOrigin,379.20,51.11,0.00),v40,fine,tPen\WObj:=wPaper;
    MoveL Offs(pOrigin,379.20,51.11,6.00),v60,z5,tPen\WObj:=wPaper;
    MoveL Offs(pOrigin,382.17,48.35,6.00),vTravel,z5,tPen\WObj:=wPaper;
    MoveL Offs(pOrigin,382.17,48.35,0.00),v60,z0,tPen\WObj:=wPaper;
    MoveL Offs(pOrigin,381.96,48.78,0.00),v40,z0,tPen\WObj:=wPaper;
    MoveL Offs(pOrigin,382.17,48.35,0.00),v40,z0,tPen\WObj:=wPaper;
    MoveL Offs(pOrigin,382.60,48.14,0.00),v40,z0,tPen\WObj:=wPaper;
    MoveL Offs(pOrigin,382.81,47.71,0.00),v40,z0,tPen\WObj:=wPaper;
    MoveL Offs(pOrigin,382.60,48.14,0.00),v40,fine,tPen\WObj:=wPaper;
    MoveL Offs(pOrigin,382.60,48.14,6.00),v60,z5,tPen\WObj:=wPaper;
    MoveL Offs(pOrigin,383.45,47.08,6.00),vTravel,z5,tPen\WObj:=wPaper;
    MoveL Offs(pOrigin,383.45,47.08,0.00),v60,z0,tPen\WObj:=wPaper;
    MoveL Offs(pOrigin,383.24,47.50,0.00),v40,z0,tPen\WObj:=wPaper;
    MoveL Offs(pOrigin,383.45,47.08,0.00),v40,fine,tPen\WObj:=wPaper;
    MoveL Offs(pOrigin,383.45,47.08,6.00),v60,z5,tPen\WObj:=wPaper;
    MoveL Offs(pOrigin,346.90,46.44,6.00),vTravel,z5,tPen\WObj:=wPaper;
    MoveL Offs(pOrigin,346.90,46.44,0.00),v60,z0,tPen\WObj:=wPaper;
    MoveL Offs(pOrigin,346.69,46.86,0.00),v40,z0,tPen\WObj:=wPaper;
    MoveL Offs(pOrigin,346.90,46.44,0.00),v40,fine,tPen\WObj:=wPaper;
    MoveL Offs(pOrigin,346.90,46.44,6.00),v60,z5,tPen\WObj:=wPaper;
    MoveL Offs(pOrigin,343.71,51.54,6.00),vTravel,z5,tPen\WObj:=wPaper;
    MoveL Offs(pOrigin,343.71,51.54,0.00),v60,z0,tPen\WObj:=wPaper;
    MoveL Offs(pOrigin,343.50,51.96,0.00),v40,z0,tPen\WObj:=wPaper;
    MoveL Offs(pOrigin,343.71,51.54,0.00),v40,fine,tPen\WObj:=wPaper;
    MoveL Offs(pOrigin,343.71,51.54,6.00),v60,z5,tPen\WObj:=wPaper;
    MoveL Offs(pOrigin,341.38,54.72,6.00),vTravel,z5,tPen\WObj:=wPaper;
    MoveL Offs(pOrigin,341.38,54.72,0.00),v60,z0,tPen\WObj:=wPaper;
    MoveL Offs(pOrigin,340.95,55.36,0.00),v40,z0,tPen\WObj:=wPaper;
    MoveL Offs(pOrigin,341.38,54.72,0.00),v40,fine,tPen\WObj:=wPaper;
    MoveL Offs(pOrigin,341.38,54.72,6.00),v60,z5,tPen\WObj:=wPaper;
    MoveL Offs(pOrigin,339.46,57.06,6.00),vTravel,z5,tPen\WObj:=wPaper;
    MoveL Offs(pOrigin,339.46,57.06,0.00),v60,z0,tPen\WObj:=wPaper;
    MoveL Offs(pOrigin,337.76,58.76,0.00),v40,z0,tPen\WObj:=wPaper;
    MoveL Offs(pOrigin,339.46,57.06,0.00),v40,fine,tPen\WObj:=wPaper;
    MoveL Offs(pOrigin,339.46,57.06,6.00),v60,z5,tPen\WObj:=wPaper;
    MoveL Offs(pOrigin,337.55,58.97,6.00),vTravel,z5,tPen\WObj:=wPaper;
    MoveL Offs(pOrigin,337.55,58.97,0.00),v60,z0,tPen\WObj:=wPaper;
    MoveL Offs(pOrigin,336.91,59.61,0.00),v40,z0,tPen\WObj:=wPaper;
    MoveL Offs(pOrigin,337.55,58.97,0.00),v40,fine,tPen\WObj:=wPaper;
    MoveL Offs(pOrigin,337.55,58.97,6.00),v60,z5,tPen\WObj:=wPaper;
    MoveL Offs(pOrigin,334.79,57.28,6.00),vTravel,z5,tPen\WObj:=wPaper;
    MoveL Offs(pOrigin,334.79,57.28,0.00),v60,z0,tPen\WObj:=wPaper;
    MoveL Offs(pOrigin,336.98,54.09,0.00),v40,z0,tPen\WObj:=wPaper;
    MoveL Offs(pOrigin,337.98,51.96,0.00),v40,fine,tPen\WObj:=wPaper;
    MoveL Offs(pOrigin,337.98,51.96,6.00),v60,z5,tPen\WObj:=wPaper;
    MoveL Offs(pOrigin,337.12,53.45,6.00),vTravel,z5,tPen\WObj:=wPaper;
    MoveL Offs(pOrigin,337.12,53.45,0.00),v60,z0,tPen\WObj:=wPaper;
    MoveL Offs(pOrigin,336.91,53.88,0.00),v40,z0,tPen\WObj:=wPaper;
    MoveL Offs(pOrigin,337.12,53.45,0.00),v40,fine,tPen\WObj:=wPaper;
    MoveL Offs(pOrigin,337.12,53.45,6.00),v60,z5,tPen\WObj:=wPaper;
    MoveL Offs(pOrigin,336.27,54.94,6.00),vTravel,z5,tPen\WObj:=wPaper;
    MoveL Offs(pOrigin,336.27,54.94,0.00),v60,z0,tPen\WObj:=wPaper;
    MoveL Offs(pOrigin,335.85,55.58,0.00),v40,z0,tPen\WObj:=wPaper;
    MoveL Offs(pOrigin,336.27,54.94,0.00),v40,fine,tPen\WObj:=wPaper;
    MoveL Offs(pOrigin,336.27,54.94,6.00),v60,z5,tPen\WObj:=wPaper;
    MoveL Offs(pOrigin,317.58,59.83,6.00),vTravel,z5,tPen\WObj:=wPaper;
    MoveL Offs(pOrigin,317.58,59.83,0.00),v60,z0,tPen\WObj:=wPaper;
    MoveL Offs(pOrigin,317.15,60.25,0.00),v40,z0,tPen\WObj:=wPaper;
    MoveL Offs(pOrigin,317.58,59.83,0.00),v40,fine,tPen\WObj:=wPaper;
    MoveL Offs(pOrigin,317.58,59.83,6.00),v60,z5,tPen\WObj:=wPaper;
    MoveL Offs(pOrigin,310.56,61.10,6.00),vTravel,z5,tPen\WObj:=wPaper;
    MoveL Offs(pOrigin,310.56,61.10,0.00),v60,z0,tPen\WObj:=wPaper;
    MoveL Offs(pOrigin,310.99,62.80,0.00),v40,fine,tPen\WObj:=wPaper;
    MoveL Offs(pOrigin,310.99,62.80,6.00),v60,z5,tPen\WObj:=wPaper;
    MoveL Offs(pOrigin,313.11,67.69,6.00),vTravel,z5,tPen\WObj:=wPaper;
    MoveL Offs(pOrigin,313.11,67.69,0.00),v60,z0,tPen\WObj:=wPaper;
    MoveL Offs(pOrigin,310.99,66.84,0.00),v40,z0,tPen\WObj:=wPaper;
    MoveL Offs(pOrigin,305.04,65.56,0.00),v40,z0,tPen\WObj:=wPaper;
    MoveL Offs(pOrigin,301.85,64.36,0.00),v40,z0,tPen\WObj:=wPaper;
    MoveL Offs(pOrigin,299.73,63.01,0.00),v40,z0,tPen\WObj:=wPaper;
    MoveL Offs(pOrigin,299.09,61.95,0.00),v40,z0,tPen\WObj:=wPaper;
    MoveL Offs(pOrigin,299.09,61.95,0.00),v40,z0,tPen\WObj:=wPaper;
    MoveL Offs(pOrigin,300.15,61.31,0.00),v40,z0,tPen\WObj:=wPaper;
    MoveL Offs(pOrigin,301.85,61.31,0.00),v40,fine,tPen\WObj:=wPaper;
    MoveL Offs(pOrigin,301.85,61.31,6.00),v60,z5,tPen\WObj:=wPaper;
    MoveL Offs(pOrigin,299.30,61.53,6.00),vTravel,z5,tPen\WObj:=wPaper;
    MoveL Offs(pOrigin,299.30,61.53,0.00),v60,z0,tPen\WObj:=wPaper;
    MoveL Offs(pOrigin,299.09,61.95,0.00),v40,z0,tPen\WObj:=wPaper;
    MoveL Offs(pOrigin,299.30,61.53,0.00),v40,z0,tPen\WObj:=wPaper;
    MoveL Offs(pOrigin,299.09,61.95,0.00),v40,z0,tPen\WObj:=wPaper;
    MoveL Offs(pOrigin,296.54,62.38,0.00),v40,z0,tPen\WObj:=wPaper;
    MoveL Offs(pOrigin,292.92,63.58,0.00),v40,z0,tPen\WObj:=wPaper;
    MoveL Offs(pOrigin,289.74,65.07,0.00),v40,z0,tPen\WObj:=wPaper;
    MoveL Offs(pOrigin,286.12,67.12,0.00),v40,z0,tPen\WObj:=wPaper;
    MoveL Offs(pOrigin,285.70,67.69,0.00),v40,fine,tPen\WObj:=wPaper;
    MoveL Offs(pOrigin,285.70,67.69,6.00),v60,z5,tPen\WObj:=wPaper;
    MoveL Offs(pOrigin,288.46,65.99,6.00),vTravel,z5,tPen\WObj:=wPaper;
    MoveL Offs(pOrigin,288.46,65.99,0.00),v60,z0,tPen\WObj:=wPaper;
    MoveL Offs(pOrigin,288.89,65.78,0.00),v40,z0,tPen\WObj:=wPaper;
    MoveL Offs(pOrigin,288.46,65.99,0.00),v40,fine,tPen\WObj:=wPaper;
    MoveL Offs(pOrigin,288.46,65.99,6.00),v60,z5,tPen\WObj:=wPaper;
    MoveL Offs(pOrigin,289.52,65.35,6.00),vTravel,z5,tPen\WObj:=wPaper;
    MoveL Offs(pOrigin,289.52,65.35,0.00),v60,z0,tPen\WObj:=wPaper;
    MoveL Offs(pOrigin,289.95,65.14,0.00),v40,z0,tPen\WObj:=wPaper;
    MoveL Offs(pOrigin,289.52,65.35,0.00),v40,z0,tPen\WObj:=wPaper;
    MoveL Offs(pOrigin,290.38,64.93,0.00),v40,z0,tPen\WObj:=wPaper;
    MoveL Offs(pOrigin,290.80,64.71,0.00),v40,z0,tPen\WObj:=wPaper;
    MoveL Offs(pOrigin,290.38,64.93,0.00),v40,fine,tPen\WObj:=wPaper;
    MoveL Offs(pOrigin,290.38,64.93,6.00),v60,z5,tPen\WObj:=wPaper;
    MoveL Offs(pOrigin,294.41,65.56,6.00),vTravel,z5,tPen\WObj:=wPaper;
    MoveL Offs(pOrigin,294.41,65.56,0.00),v60,z0,tPen\WObj:=wPaper;
    MoveL Offs(pOrigin,293.56,68.54,0.00),v40,z0,tPen\WObj:=wPaper;
    MoveL Offs(pOrigin,292.29,77.46,0.00),v40,z0,tPen\WObj:=wPaper;
    MoveL Offs(pOrigin,292.08,91.70,0.00),v40,z0,tPen\WObj:=wPaper;
    MoveL Offs(pOrigin,292.50,97.22,0.00),v40,z0,tPen\WObj:=wPaper;
    MoveL Offs(pOrigin,291.86,98.07,0.00),v40,z0,tPen\WObj:=wPaper;
    MoveL Offs(pOrigin,291.86,98.07,0.00),v40,z0,tPen\WObj:=wPaper;
    MoveL Offs(pOrigin,291.37,97.44,0.00),v40,z0,tPen\WObj:=wPaper;
    MoveL Offs(pOrigin,287.61,81.50,0.00),v40,z0,tPen\WObj:=wPaper;
    MoveL Offs(pOrigin,285.49,67.76,0.00),v40,z0,tPen\WObj:=wPaper;
    MoveL Offs(pOrigin,281.88,67.90,0.00),v40,z0,tPen\WObj:=wPaper;
    MoveL Offs(pOrigin,275.71,65.78,0.00),v40,z0,tPen\WObj:=wPaper;
    MoveL Offs(pOrigin,275.29,65.99,0.00),v40,z0,tPen\WObj:=wPaper;
    MoveL Offs(pOrigin,272.74,80.44,0.00),v40,z0,tPen\WObj:=wPaper;
  ENDPROC

